   1:L PR[91] 10mm/sec FINE;
   1:  PR[GP1:91,1] = PR[GP1:90,1] + 93.609;
   1:  PR[GP1:91,2] = PR[GP1:90,2] + 108.231;
   1:L PR[91] 10mm/sec FINE;
   1:  PR[GP1:91,1] = PR[GP1:90,1] + 93.731;
   1:  PR[GP1:91,2] = PR[GP1:90,2] + 108.362;
   1:L PR[91] 10mm/sec FINE;
   1:  PR[GP1:91,1] = PR[GP1:90,1] + 93.913;
   1:  PR[GP1:91,2] = PR[GP1:90,2] + 108.511;
   1:L PR[91] 10mm/sec FINE;
   1:  PR[GP1:91,1] = PR[GP1:90,1] + 94.171;
   1:  PR[GP1:91,2] = PR[GP1:90,2] + 108.665;
   1:L PR[91] 10mm/sec FINE;
   1:  PR[GP1:91,1] = PR[GP1:90,1] + 94.322;
   1:  PR[GP1:91,2] = PR[GP1:90,2] + 108.701;
   1:L PR[91] 10mm/sec FINE;
   1:  PR[GP1:91,1] = PR[GP1:90,1] + 94.513;
   1:  PR[GP1:91,2] = PR[GP1:90,2] + 108.801;
   1:L PR[91] 10mm/sec FINE;
   1:  PR[GP1:91,1] = PR[GP1:90,1] + 94.701;
   1:  PR[GP1:91,2] = PR[GP1:90,2] + 108.857;
   1:L PR[91] 10mm/sec FINE;
   1:  PR[GP1:91,1] = PR[GP1:90,1] + 94.821;
   1:  PR[GP1:91,2] = PR[GP1:90,2] + 108.845;
   1:L PR[91] 10mm/sec FINE;
   1:  PR[GP1:91,1] = PR[GP1:90,1] + 95.615;
   1:  PR[GP1:91,2] = PR[GP1:90,2] + 108.874;
   1:L PR[91] 10mm/sec FINE;
   1:  PR[GP1:91,1] = PR[GP1:90,1] + 95.743;
   1:  PR[GP1:91,2] = PR[GP1:90,2] + 108.844;
   1:L PR[91] 10mm/sec FINE;
   1:  PR[GP1:91,1] = PR[GP1:90,1] + 96.602;
   1:  PR[GP1:91,2] = PR[GP1:90,2] + 108.491;
   1:L PR[91] 10mm/sec FINE;
   1:  PR[GP1:91,1] = PR[GP1:90,1] + 96.918;
   1:  PR[GP1:91,2] = PR[GP1:90,2] + 108.237;
   1:L PR[91] 10mm/sec FINE;
   1:  PR[GP1:91,1] = PR[GP1:90,1] + 97.426;
   1:  PR[GP1:91,2] = PR[GP1:90,2] + 107.738;
   1:L PR[91] 10mm/sec FINE;
   1:  PR[GP1:91,1] = PR[GP1:90,1] + 97.882;
   1:  PR[GP1:91,2] = PR[GP1:90,2] + 106.699;
   1:L PR[91] 10mm/sec FINE;
   1:  PR[GP1:91,1] = PR[GP1:90,1] + 98.569;
   1:  PR[GP1:91,2] = PR[GP1:90,2] + 104.056;
   1:L PR[91] 10mm/sec FINE;
   1:  PR[GP1:91,1] = PR[GP1:90,1] + 99.310;
   1:  PR[GP1:91,2] = PR[GP1:90,2] + 102.392;
   1:L PR[91] 10mm/sec FINE;
   1:  PR[GP1:91,1] = PR[GP1:90,1] + 99.684;
   1:  PR[GP1:91,2] = PR[GP1:90,2] + 101.561;
   1:L PR[91] 10mm/sec FINE;
   1:  PR[GP1:91,1] = PR[GP1:90,1] + 101.201;
   1:  PR[GP1:91,2] = PR[GP1:90,2] + 99.269;
   1:L PR[91] 10mm/sec FINE;
   1:  PR[GP1:91,1] = PR[GP1:90,1] + 103.078;
   1:  PR[GP1:91,2] = PR[GP1:90,2] + 97.241;
   1:L PR[91] 10mm/sec FINE;
   1:  PR[GP1:91,1] = PR[GP1:90,1] + 105.216;
   1:  PR[GP1:91,2] = PR[GP1:90,2] + 95.523;
   1:L PR[91] 10mm/sec FINE;
   1:  PR[GP1:91,1] = PR[GP1:90,1] + 107.581;
   1:  PR[GP1:91,2] = PR[GP1:90,2] + 94.152;
   1:L PR[91] 10mm/sec FINE;
   1:  PR[GP1:91,1] = PR[GP1:90,1] + 110.132;
   1:  PR[GP1:91,2] = PR[GP1:90,2] + 93.162;
   1:L PR[91] 10mm/sec FINE;
   1:  PR[GP1:91,1] = PR[GP1:90,1] + 112.809;
   1:  PR[GP1:91,2] = PR[GP1:90,2] + 92.574;
   1:L PR[91] 10mm/sec FINE;
   1:  PR[GP1:91,1] = PR[GP1:90,1] + 115.553;
   1:  PR[GP1:91,2] = PR[GP1:90,2] + 92.397;
   1:L PR[91] 10mm/sec FINE;
   1:  PR[GP1:91,1] = PR[GP1:90,1] + 118.148;
   1:  PR[GP1:91,2] = PR[GP1:90,2] + 92.625;
   1:L PR[91] 10mm/sec FINE;
   1:  PR[GP1:91,1] = PR[GP1:90,1] + 118.473;
   1:  PR[GP1:91,2] = PR[GP1:90,2] + 92.690;
   1:L PR[91] 10mm/sec FINE;
   1:  PR[GP1:91,1] = PR[GP1:90,1] + 120.533;
   1:  PR[GP1:91,2] = PR[GP1:90,2] + 93.200;
   1:L PR[91] 10mm/sec FINE;
   1:  PR[GP1:91,1] = PR[GP1:90,1] + 121.008;
   1:  PR[GP1:91,2] = PR[GP1:90,2] + 93.351;
   1:L PR[91] 10mm/sec FINE;
   1:  PR[GP1:91,1] = PR[GP1:90,1] + 123.294;
   1:  PR[GP1:91,2] = PR[GP1:90,2] + 94.329;
   1:L PR[91] 10mm/sec FINE;
   1:  PR[GP1:91,1] = PR[GP1:90,1] + 123.840;
   1:  PR[GP1:91,2] = PR[GP1:90,2] + 94.647;
   1:L PR[91] 10mm/sec FINE;
   1:  PR[GP1:91,1] = PR[GP1:90,1] + 125.327;
   1:  PR[GP1:91,2] = PR[GP1:90,2] + 95.571;
   1:L PR[91] 10mm/sec FINE;
   1:  PR[GP1:91,1] = PR[GP1:90,1] + 125.920;
   1:  PR[GP1:91,2] = PR[GP1:90,2] + 96.009;
   1:L PR[91] 10mm/sec FINE;
   1:  PR[GP1:91,1] = PR[GP1:90,1] + 127.113;
   1:  PR[GP1:91,2] = PR[GP1:90,2] + 97.040;
   1:L PR[91] 10mm/sec FINE;
   1:  PR[GP1:91,1] = PR[GP1:90,1] + 127.715;
   1:  PR[GP1:91,2] = PR[GP1:90,2] + 97.597;
   1:L PR[91] 10mm/sec FINE;
   1:  PR[GP1:91,1] = PR[GP1:90,1] + 129.232;
   1:  PR[GP1:91,2] = PR[GP1:90,2] + 99.375;
   1:L PR[91] 10mm/sec FINE;
   1:  PR[GP1:91,1] = PR[GP1:90,1] + 129.733;
   1:  PR[GP1:91,2] = PR[GP1:90,2] + 100.102;
   1:L PR[91] 10mm/sec FINE;
   1:  PR[GP1:91,1] = PR[GP1:90,1] + 130.464;
   1:  PR[GP1:91,2] = PR[GP1:90,2] + 101.304;
   1:L PR[91] 10mm/sec FINE;
   1:  PR[GP1:91,1] = PR[GP1:90,1] + 130.906;
   1:  PR[GP1:91,2] = PR[GP1:90,2] + 102.124;
   1:L PR[91] 10mm/sec FINE;
   1:  PR[GP1:91,1] = PR[GP1:90,1] + 131.776;
   1:  PR[GP1:91,2] = PR[GP1:90,2] + 104.258;
   1:L PR[91] 10mm/sec FINE;
   1:  PR[GP1:91,1] = PR[GP1:90,1] + 132.039;
   1:  PR[GP1:91,2] = PR[GP1:90,2] + 105.190;
   1:L PR[91] 10mm/sec FINE;
   1:  PR[GP1:91,1] = PR[GP1:90,1] + 132.341;
   1:  PR[GP1:91,2] = PR[GP1:90,2] + 106.462;
   1:L PR[91] 10mm/sec FINE;
   1:  PR[GP1:91,1] = PR[GP1:90,1] + 132.504;
   1:  PR[GP1:91,2] = PR[GP1:90,2] + 107.439;
   1:L PR[91] 10mm/sec FINE;
   1:  PR[GP1:91,1] = PR[GP1:90,1] + 132.559;
   1:  PR[GP1:91,2] = PR[GP1:90,2] + 108.440;
   1:L PR[91] 10mm/sec FINE;
   1:  PR[GP1:91,1] = PR[GP1:90,1] + 132.683;
   1:  PR[GP1:91,2] = PR[GP1:90,2] + 109.720;
   1:L PR[91] 10mm/sec FINE;
   1:  PR[GP1:91,1] = PR[GP1:90,1] + 132.328;
   1:  PR[GP1:91,2] = PR[GP1:90,2] + 113.118;
   1:L PR[91] 10mm/sec FINE;
   1:  PR[GP1:91,1] = PR[GP1:90,1] + 131.820;
   1:  PR[GP1:91,2] = PR[GP1:90,2] + 114.773;
   1:L PR[91] 10mm/sec FINE;
   1:  PR[GP1:91,1] = PR[GP1:90,1] + 131.524;
   1:  PR[GP1:91,2] = PR[GP1:90,2] + 115.868;
   1:L PR[91] 10mm/sec FINE;
   1:  PR[GP1:91,1] = PR[GP1:90,1] + 131.329;
   1:  PR[GP1:91,2] = PR[GP1:90,2] + 116.382;
   1:L PR[91] 10mm/sec FINE;
   1:  PR[GP1:91,1] = PR[GP1:90,1] + 129.702;
   1:  PR[GP1:91,2] = PR[GP1:90,2] + 119.396;
   1:L PR[91] 10mm/sec FINE;
   1:  PR[GP1:91,1] = PR[GP1:90,1] + 128.498;
   1:  PR[GP1:91,2] = PR[GP1:90,2] + 120.846;
   1:L PR[91] 10mm/sec FINE;
   1:  PR[GP1:91,1] = PR[GP1:90,1] + 128.197;
   1:  PR[GP1:91,2] = PR[GP1:90,2] + 121.262;
   1:L PR[91] 10mm/sec FINE;
   1:  PR[GP1:91,1] = PR[GP1:90,1] + 127.521;
   1:  PR[GP1:91,2] = PR[GP1:90,2] + 122.025;
   1:L PR[91] 10mm/sec FINE;
   1:  PR[GP1:91,1] = PR[GP1:90,1] + 124.860;
   1:  PR[GP1:91,2] = PR[GP1:90,2] + 124.177;
   1:L PR[91] 10mm/sec FINE;
   1:  PR[GP1:91,1] = PR[GP1:90,1] + 121.833;
   1:  PR[GP1:91,2] = PR[GP1:90,2] + 125.763;
   1:L PR[91] 10mm/sec FINE;
   1:  PR[GP1:91,1] = PR[GP1:90,1] + 119.391;
   1:  PR[GP1:91,2] = PR[GP1:90,2] + 126.477;
   1:L PR[91] 10mm/sec FINE;
   1:  PR[GP1:91,1] = PR[GP1:90,1] + 118.835;
   1:  PR[GP1:91,2] = PR[GP1:90,2] + 126.660;
   1:L PR[91] 10mm/sec FINE;
   1:  PR[GP1:91,1] = PR[GP1:90,1] + 118.561;
   1:  PR[GP1:91,2] = PR[GP1:90,2] + 126.721;
   1:L PR[91] 10mm/sec FINE;
   1:  PR[GP1:91,1] = PR[GP1:90,1] + 115.143;
   1:  PR[GP1:91,2] = PR[GP1:90,2] + 127.017;
   1:L PR[91] 10mm/sec FINE;
   1:  PR[GP1:91,1] = PR[GP1:90,1] + 111.751;
   1:  PR[GP1:91,2] = PR[GP1:90,2] + 126.637;
   1:L PR[91] 10mm/sec FINE;
   1:  PR[GP1:91,1] = PR[GP1:90,1] + 108.452;
   1:  PR[GP1:91,2] = PR[GP1:90,2] + 125.593;
   1:L PR[91] 10mm/sec FINE;
   1:  PR[GP1:91,1] = PR[GP1:90,1] + 105.418;
   1:  PR[GP1:91,2] = PR[GP1:90,2] + 123.928;
   1:L PR[91] 10mm/sec FINE;
   1:  PR[GP1:91,1] = PR[GP1:90,1] + 102.775;
   1:  PR[GP1:91,2] = PR[GP1:90,2] + 121.709;
   1:L PR[91] 10mm/sec FINE;
   1:  PR[GP1:91,1] = PR[GP1:90,1] + 100.581;
   1:  PR[GP1:91,2] = PR[GP1:90,2] + 119.016;
   1:L PR[91] 10mm/sec FINE;
   1:  PR[GP1:91,1] = PR[GP1:90,1] + 98.955;
   1:  PR[GP1:91,2] = PR[GP1:90,2] + 115.958;
   1:L PR[91] 10mm/sec FINE;
   1:  PR[GP1:91,1] = PR[GP1:90,1] + 97.961;
   1:  PR[GP1:91,2] = PR[GP1:90,2] + 112.694;
   1:L PR[91] 10mm/sec FINE;
   1:  PR[GP1:91,1] = PR[GP1:90,1] + 97.646;
   1:  PR[GP1:91,2] = PR[GP1:90,2] + 112.056;
   1:L PR[91] 10mm/sec FINE;
   1:  PR[GP1:91,1] = PR[GP1:90,1] + 97.480;
   1:  PR[GP1:91,2] = PR[GP1:90,2] + 111.669;
   1:L PR[91] 10mm/sec FINE;
   1:  PR[GP1:91,1] = PR[GP1:90,1] + 97.077;
   1:  PR[GP1:91,2] = PR[GP1:90,2] + 111.285;
   1:L PR[91] 10mm/sec FINE;
   1:  PR[GP1:91,1] = PR[GP1:90,1] + 96.627;
   1:  PR[GP1:91,2] = PR[GP1:90,2] + 110.927;
   1:L PR[91] 10mm/sec FINE;
   1:  PR[GP1:91,1] = PR[GP1:90,1] + 95.953;
   1:  PR[GP1:91,2] = PR[GP1:90,2] + 110.656;
   1:L PR[91] 10mm/sec FINE;
   1:  PR[GP1:91,1] = PR[GP1:90,1] + 95.474;
   1:  PR[GP1:91,2] = PR[GP1:90,2] + 110.548;
   1:L PR[91] 10mm/sec FINE;
   1:  PR[GP1:91,1] = PR[GP1:90,1] + 94.864;
   1:  PR[GP1:91,2] = PR[GP1:90,2] + 110.569;
   1:L PR[91] 10mm/sec FINE;
   1:  PR[GP1:91,1] = PR[GP1:90,1] + 94.445;
   1:  PR[GP1:91,2] = PR[GP1:90,2] + 110.680;
   1:L PR[91] 10mm/sec FINE;
   1:  PR[GP1:91,1] = PR[GP1:90,1] + 94.027;
   1:  PR[GP1:91,2] = PR[GP1:90,2] + 110.868;
   1:L PR[91] 10mm/sec FINE;
   1:  PR[GP1:91,1] = PR[GP1:90,1] + 93.791;
   1:  PR[GP1:91,2] = PR[GP1:90,2] + 111.065;
   1:L PR[91] 10mm/sec FINE;
   1:  PR[GP1:91,1] = PR[GP1:90,1] + 93.574;
   1:  PR[GP1:91,2] = PR[GP1:90,2] + 111.221;
   1:L PR[91] 10mm/sec FINE;
   1:  PR[GP1:91,1] = PR[GP1:90,1] + 93.370;
   1:  PR[GP1:91,2] = PR[GP1:90,2] + 111.406;
   1:L PR[91] 10mm/sec FINE;
   1:  PR[GP1:91,1] = PR[GP1:90,1] + 93.152;
   1:  PR[GP1:91,2] = PR[GP1:90,2] + 111.677;
   1:L PR[91] 10mm/sec FINE;
   1:  PR[GP1:91,1] = PR[GP1:90,1] + 92.966;
   1:  PR[GP1:91,2] = PR[GP1:90,2] + 112.106;
   1:L PR[91] 10mm/sec FINE;
   1:  PR[GP1:91,1] = PR[GP1:90,1] + 92.851;
   1:  PR[GP1:91,2] = PR[GP1:90,2] + 112.318;
   1:L PR[91] 10mm/sec FINE;
   1:  PR[GP1:91,1] = PR[GP1:90,1] + 92.770;
   1:  PR[GP1:91,2] = PR[GP1:90,2] + 112.528;
   1:L PR[91] 10mm/sec FINE;
   1:  PR[GP1:91,1] = PR[GP1:90,1] + 92.754;
   1:  PR[GP1:91,2] = PR[GP1:90,2] + 112.593;
   1:L PR[91] 10mm/sec FINE;
   1:  PR[GP1:91,1] = PR[GP1:90,1] + 92.675;
   1:  PR[GP1:91,2] = PR[GP1:90,2] + 112.597;
   1:L PR[91] 10mm/sec FINE;
   1:  PR[GP1:91,1] = PR[GP1:90,1] + 92.473;
   1:  PR[GP1:91,2] = PR[GP1:90,2] + 113.514;
   1:L PR[91] 10mm/sec FINE;
   1:  PR[GP1:91,1] = PR[GP1:90,1] + 91.748;
   1:  PR[GP1:91,2] = PR[GP1:90,2] + 116.014;
   1:L PR[91] 10mm/sec FINE;
   1:  PR[GP1:91,1] = PR[GP1:90,1] + 91.367;
   1:  PR[GP1:91,2] = PR[GP1:90,2] + 116.861;
   1:L PR[91] 10mm/sec FINE;
   1:  PR[GP1:91,1] = PR[GP1:90,1] + 90.243;
   1:  PR[GP1:91,2] = PR[GP1:90,2] + 118.946;
   1:L PR[91] 10mm/sec FINE;
   1:  PR[GP1:91,1] = PR[GP1:90,1] + 89.639;
   1:  PR[GP1:91,2] = PR[GP1:90,2] + 119.852;
   1:L PR[91] 10mm/sec FINE;
   1:  PR[GP1:91,1] = PR[GP1:90,1] + 88.262;
   1:  PR[GP1:91,2] = PR[GP1:90,2] + 121.466;
   1:L PR[91] 10mm/sec FINE;
   1:  PR[GP1:91,1] = PR[GP1:90,1] + 87.411;
   1:  PR[GP1:91,2] = PR[GP1:90,2] + 122.375;
   1:L PR[91] 10mm/sec FINE;
   1:  PR[GP1:91,1] = PR[GP1:90,1] + 84.803;
   1:  PR[GP1:91,2] = PR[GP1:90,2] + 124.368;
   1:L PR[91] 10mm/sec FINE;
   1:  PR[GP1:91,1] = PR[GP1:90,1] + 83.575;
   1:  PR[GP1:91,2] = PR[GP1:90,2] + 125.021;
   1:L PR[91] 10mm/sec FINE;
   1:  PR[GP1:91,1] = PR[GP1:90,1] + 81.935;
   1:  PR[GP1:91,2] = PR[GP1:90,2] + 125.795;
   1:L PR[91] 10mm/sec FINE;
   1:  PR[GP1:91,1] = PR[GP1:90,1] + 80.497;
   1:  PR[GP1:91,2] = PR[GP1:90,2] + 126.278;
   1:L PR[91] 10mm/sec FINE;
   1:  PR[GP1:91,1] = PR[GP1:90,1] + 78.911;
   1:  PR[GP1:91,2] = PR[GP1:90,2] + 126.649;
   1:L PR[91] 10mm/sec FINE;
   1:  PR[GP1:91,1] = PR[GP1:90,1] + 77.310;
   1:  PR[GP1:91,2] = PR[GP1:90,2] + 126.906;
   1:L PR[91] 10mm/sec FINE;
   1:  PR[GP1:91,1] = PR[GP1:90,1] + 75.679;
   1:  PR[GP1:91,2] = PR[GP1:90,2] + 126.897;
   1:L PR[91] 10mm/sec FINE;
   1:  PR[GP1:91,1] = PR[GP1:90,1] + 74.111;
   1:  PR[GP1:91,2] = PR[GP1:90,2] + 126.922;
   1:L PR[91] 10mm/sec FINE;
   1:  PR[GP1:91,1] = PR[GP1:90,1] + 72.423;
   1:  PR[GP1:91,2] = PR[GP1:90,2] + 126.632;
   1:L PR[91] 10mm/sec FINE;
   1:  PR[GP1:91,1] = PR[GP1:90,1] + 71.016;
   1:  PR[GP1:91,2] = PR[GP1:90,2] + 126.355;
   1:L PR[91] 10mm/sec FINE;
   1:  PR[GP1:91,1] = PR[GP1:90,1] + 69.332;
   1:  PR[GP1:91,2] = PR[GP1:90,2] + 125.768;
   1:L PR[91] 10mm/sec FINE;
   1:  PR[GP1:91,1] = PR[GP1:90,1] + 68.107;
   1:  PR[GP1:91,2] = PR[GP1:90,2] + 125.242;
   1:L PR[91] 10mm/sec FINE;
   1:  PR[GP1:91,1] = PR[GP1:90,1] + 66.494;
   1:  PR[GP1:91,2] = PR[GP1:90,2] + 124.361;
   1:L PR[91] 10mm/sec FINE;
   1:  PR[GP1:91,1] = PR[GP1:90,1] + 65.466;
   1:  PR[GP1:91,2] = PR[GP1:90,2] + 123.631;
   1:L PR[91] 10mm/sec FINE;
   1:  PR[GP1:91,1] = PR[GP1:90,1] + 63.989;
   1:  PR[GP1:91,2] = PR[GP1:90,2] + 122.474;
   1:L PR[91] 10mm/sec FINE;
   1:  PR[GP1:91,1] = PR[GP1:90,1] + 61.881;
   1:  PR[GP1:91,2] = PR[GP1:90,2] + 120.170;
   1:L PR[91] 10mm/sec FINE;
   1:  PR[GP1:91,1] = PR[GP1:90,1] + 60.844;
   1:  PR[GP1:91,2] = PR[GP1:90,2] + 118.575;
   1:L PR[91] 10mm/sec FINE;
   1:  PR[GP1:91,1] = PR[GP1:90,1] + 60.235;
   1:  PR[GP1:91,2] = PR[GP1:90,2] + 117.535;
   1:L PR[91] 10mm/sec FINE;
   1:  PR[GP1:91,1] = PR[GP1:90,1] + 59.468;
   1:  PR[GP1:91,2] = PR[GP1:90,2] + 115.779;
   1:L PR[91] 10mm/sec FINE;
   1:  PR[GP1:91,1] = PR[GP1:90,1] + 59.094;
   1:  PR[GP1:91,2] = PR[GP1:90,2] + 114.645;
   1:L PR[91] 10mm/sec FINE;
   1:  PR[GP1:91,1] = PR[GP1:90,1] + 58.626;
   1:  PR[GP1:91,2] = PR[GP1:90,2] + 112.789;
   1:L PR[91] 10mm/sec FINE;
   1:  PR[GP1:91,1] = PR[GP1:90,1] + 58.468;
   1:  PR[GP1:91,2] = PR[GP1:90,2] + 110.872;
   1:L PR[91] 10mm/sec FINE;
   1:  PR[GP1:91,1] = PR[GP1:90,1] + 58.343;
   1:  PR[GP1:91,2] = PR[GP1:90,2] + 109.685;
   1:L PR[91] 10mm/sec FINE;
   1:  PR[GP1:91,1] = PR[GP1:90,1] + 58.500;
   1:  PR[GP1:91,2] = PR[GP1:90,2] + 107.787;
   1:L PR[91] 10mm/sec FINE;
   1:  PR[GP1:91,1] = PR[GP1:90,1] + 58.630;
   1:  PR[GP1:91,2] = PR[GP1:90,2] + 106.576;
   1:L PR[91] 10mm/sec FINE;
   1:  PR[GP1:91,1] = PR[GP1:90,1] + 59.091;
   1:  PR[GP1:91,2] = PR[GP1:90,2] + 104.751;
   1:L PR[91] 10mm/sec FINE;
   1:  PR[GP1:91,1] = PR[GP1:90,1] + 59.485;
   1:  PR[GP1:91,2] = PR[GP1:90,2] + 103.554;
   1:L PR[91] 10mm/sec FINE;
   1:  PR[GP1:91,1] = PR[GP1:90,1] + 60.223;
   1:  PR[GP1:91,2] = PR[GP1:90,2] + 101.864;
   1:L PR[91] 10mm/sec FINE;
   1:  PR[GP1:91,1] = PR[GP1:90,1] + 60.899;
   1:  PR[GP1:91,2] = PR[GP1:90,2] + 100.714;
   1:L PR[91] 10mm/sec FINE;
   1:  PR[GP1:91,1] = PR[GP1:90,1] + 61.876;
   1:  PR[GP1:91,2] = PR[GP1:90,2] + 99.212;
   1:L PR[91] 10mm/sec FINE;
   1:  PR[GP1:91,1] = PR[GP1:90,1] + 64.014;
   1:  PR[GP1:91,2] = PR[GP1:90,2] + 96.881;
   1:L PR[91] 10mm/sec FINE;
   1:  PR[GP1:91,1] = PR[GP1:90,1] + 65.370;
   1:  PR[GP1:91,2] = PR[GP1:90,2] + 95.818;
   1:L PR[91] 10mm/sec FINE;
   1:  PR[GP1:91,1] = PR[GP1:90,1] + 66.580;
   1:  PR[GP1:91,2] = PR[GP1:90,2] + 94.963;
   1:L PR[91] 10mm/sec FINE;
   1:  PR[GP1:91,1] = PR[GP1:90,1] + 67.818;
   1:  PR[GP1:91,2] = PR[GP1:90,2] + 94.288;
   1:  PR[GP1:91,3] = PR[GP1:90,3] + 7.900;
   1:L PR[91] 10mm/sec FINE;
   1:  PR[GP1:91,1] = PR[GP1:90,1] + 69.950;
   1:  PR[GP1:91,2] = PR[GP1:90,2] + 93.380;
   1:L PR[91] 10mm/sec FINE;
   1:  PR[GP1:91,1] = PR[GP1:90,1] + 70.874;
   1:  PR[GP1:91,2] = PR[GP1:90,2] + 93.058;
   1:L PR[91] 10mm/sec FINE;
   1:  PR[GP1:91,1] = PR[GP1:90,1] + 71.846;
   1:  PR[GP1:91,2] = PR[GP1:90,2] + 92.891;
   1:L PR[91] 10mm/sec FINE;
   1:  PR[GP1:91,1] = PR[GP1:90,1] + 74.204;
   1:  PR[GP1:91,2] = PR[GP1:90,2] + 92.431;
   1:L PR[91] 10mm/sec FINE;
   1:  PR[GP1:91,1] = PR[GP1:90,1] + 75.008;
   1:  PR[GP1:91,2] = PR[GP1:90,2] + 92.426;
   1:L PR[91] 10mm/sec FINE;
   1:  PR[GP1:91,1] = PR[GP1:90,1] + 77.695;
   1:  PR[GP1:91,2] = PR[GP1:90,2] + 92.483;
   1:L PR[91] 10mm/sec FINE;
   1:  PR[GP1:91,1] = PR[GP1:90,1] + 78.289;
   1:  PR[GP1:91,2] = PR[GP1:90,2] + 92.578;
   1:L PR[91] 10mm/sec FINE;
   1:  PR[GP1:91,1] = PR[GP1:90,1] + 81.225;
   1:  PR[GP1:91,2] = PR[GP1:90,2] + 93.278;
   1:L PR[91] 10mm/sec FINE;
   1:  PR[GP1:91,1] = PR[GP1:90,1] + 81.585;
   1:  PR[GP1:91,2] = PR[GP1:90,2] + 93.398;
   1:L PR[91] 10mm/sec FINE;
   1:  PR[GP1:91,1] = PR[GP1:90,1] + 84.766;
   1:  PR[GP1:91,2] = PR[GP1:90,2] + 94.925;
   1:L PR[91] 10mm/sec FINE;
   1:  PR[GP1:91,1] = PR[GP1:90,1] + 87.670;
   1:  PR[GP1:91,2] = PR[GP1:90,2] + 97.160;
   1:L PR[91] 10mm/sec FINE;
   1:  PR[GP1:91,1] = PR[GP1:90,1] + 89.969;
   1:  PR[GP1:91,2] = PR[GP1:90,2] + 99.834;
   1:L PR[91] 10mm/sec FINE;
   1:  PR[GP1:91,1] = PR[GP1:90,1] + 90.094;
   1:  PR[GP1:91,2] = PR[GP1:90,2] + 100.009;
   1:L PR[91] 10mm/sec FINE;
   1:  PR[GP1:91,1] = PR[GP1:90,1] + 91.694;
   1:  PR[GP1:91,2] = PR[GP1:90,2] + 102.974;
   1:L PR[91] 10mm/sec FINE;
   1:  PR[GP1:91,1] = PR[GP1:90,1] + 91.822;
   1:  PR[GP1:91,2] = PR[GP1:90,2] + 103.264;
   1:L PR[91] 10mm/sec FINE;
   1:  PR[GP1:91,1] = PR[GP1:90,1] + 92.742;
   1:  PR[GP1:91,2] = PR[GP1:90,2] + 106.472;
   1:L PR[91] 10mm/sec FINE;
   1:  PR[GP1:91,1] = PR[GP1:90,1] + 92.815;
   1:  PR[GP1:91,2] = PR[GP1:90,2] + 106.821;
   1:L PR[91] 10mm/sec FINE;
   1:  PR[GP1:91,1] = PR[GP1:90,1] + 92.862;
   1:  PR[GP1:91,2] = PR[GP1:90,2] + 106.963;
   1:L PR[91] 10mm/sec FINE;
   1:  PR[GP1:91,1] = PR[GP1:90,1] + 92.947;
   1:  PR[GP1:91,2] = PR[GP1:90,2] + 107.131;
   1:L PR[91] 10mm/sec FINE;
   1:  PR[GP1:91,1] = PR[GP1:90,1] + 93.041;
   1:  PR[GP1:91,2] = PR[GP1:90,2] + 107.401;
   1:L PR[91] 10mm/sec FINE;
   1:  PR[GP1:91,1] = PR[GP1:90,1] + 93.208;
   1:  PR[GP1:91,2] = PR[GP1:90,2] + 107.720;
   1:L PR[91] 10mm/sec FINE;
   1:  PR[GP1:91,1] = PR[GP1:90,1] + 93.446;
   1:  PR[GP1:91,2] = PR[GP1:90,2] + 108.039;
   1:L PR[91] 10mm/sec FINE;
   1:  PR[GP1:91,1] = PR[GP1:90,1] + 93.610;
   1:  PR[GP1:91,2] = PR[GP1:90,2] + 108.199;
   1:L PR[91] 10mm/sec FINE;
   1:  PR[GP1:91,1] = PR[GP1:90,1] + 93.786;
   1:  PR[GP1:91,2] = PR[GP1:90,2] + 108.282;
   1:L PR[91] 10mm/sec FINE;
   1:  PR[GP1:91,1] = PR[GP1:90,1] + 94.370;
   1:  PR[GP1:91,2] = PR[GP1:90,2] + 108.653;
   1:L PR[91] 10mm/sec FINE;
   1:  PR[GP1:91,1] = PR[GP1:90,1] + 94.818;
   1:  PR[GP1:91,2] = PR[GP1:90,2] + 108.692;
   1:L PR[91] 10mm/sec FINE;
   1:  PR[GP1:91,1] = PR[GP1:90,1] + 95.314;
   1:  PR[GP1:91,2] = PR[GP1:90,2] + 108.764;
   1:L PR[91] 10mm/sec FINE;
   1:  PR[GP1:91,1] = PR[GP1:90,1] + 95.891;
   1:  PR[GP1:91,2] = PR[GP1:90,2] + 108.587;
   1:L PR[91] 10mm/sec FINE;
   1:  PR[GP1:91,1] = PR[GP1:90,1] + 96.258;
   1:  PR[GP1:91,2] = PR[GP1:90,2] + 108.434;
   1:L PR[91] 10mm/sec FINE;
   1:  PR[GP1:91,1] = PR[GP1:90,1] + 96.430;
   1:  PR[GP1:91,2] = PR[GP1:90,2] + 108.316;
   1:L PR[91] 10mm/sec FINE;
   1:  PR[GP1:91,1] = PR[GP1:90,1] + 96.886;
   1:  PR[GP1:91,2] = PR[GP1:90,2] + 107.867;
   1:L PR[91] 10mm/sec FINE;
   1:  PR[GP1:91,1] = PR[GP1:90,1] + 97.040;
   1:  PR[GP1:91,2] = PR[GP1:90,2] + 107.686;
   1:L PR[91] 10mm/sec FINE;
   1:  PR[GP1:91,1] = PR[GP1:90,1] + 97.119;
   1:  PR[GP1:91,2] = PR[GP1:90,2] + 107.556;
   1:L PR[91] 10mm/sec FINE;
   1:  PR[GP1:91,1] = PR[GP1:90,1] + 97.419;
   1:  PR[GP1:91,2] = PR[GP1:90,2] + 106.817;
   1:L PR[91] 10mm/sec FINE;
   1:  PR[GP1:91,1] = PR[GP1:90,1] + 98.137;
   1:  PR[GP1:91,2] = PR[GP1:90,2] + 104.025;
   1:L PR[91] 10mm/sec FINE;
   1:  PR[GP1:91,1] = PR[GP1:90,1] + 99.268;
   1:  PR[GP1:91,2] = PR[GP1:90,2] + 101.523;
   1:L PR[91] 10mm/sec FINE;
   1:  PR[GP1:91,1] = PR[GP1:90,1] + 100.820;
   1:  PR[GP1:91,2] = PR[GP1:90,2] + 99.224;
   1:L PR[91] 10mm/sec FINE;
   1:  PR[GP1:91,1] = PR[GP1:90,1] + 102.722;
   1:  PR[GP1:91,2] = PR[GP1:90,2] + 97.186;
   1:L PR[91] 10mm/sec FINE;
   1:  PR[GP1:91,1] = PR[GP1:90,1] + 104.917;
   1:  PR[GP1:91,2] = PR[GP1:90,2] + 95.464;
   1:L PR[91] 10mm/sec FINE;
   1:  PR[GP1:91,1] = PR[GP1:90,1] + 107.364;
   1:  PR[GP1:91,2] = PR[GP1:90,2] + 94.099;
   1:L PR[91] 10mm/sec FINE;
   1:  PR[GP1:91,1] = PR[GP1:90,1] + 109.942;
   1:  PR[GP1:91,2] = PR[GP1:90,2] + 93.112;
   1:L PR[91] 10mm/sec FINE;
   1:  PR[GP1:91,1] = PR[GP1:90,1] + 112.624;
   1:  PR[GP1:91,2] = PR[GP1:90,2] + 92.526;
   1:L PR[91] 10mm/sec FINE;
   1:  PR[GP1:91,1] = PR[GP1:90,1] + 115.365;
   1:  PR[GP1:91,2] = PR[GP1:90,2] + 92.357;
   1:L PR[91] 10mm/sec FINE;
   1:  PR[GP1:91,1] = PR[GP1:90,1] + 118.099;
   1:  PR[GP1:91,2] = PR[GP1:90,2] + 92.608;
   1:L PR[91] 10mm/sec FINE;
   1:  PR[GP1:91,1] = PR[GP1:90,1] + 120.762;
   1:  PR[GP1:91,2] = PR[GP1:90,2] + 93.274;
   1:L PR[91] 10mm/sec FINE;
   1:  PR[GP1:91,1] = PR[GP1:90,1] + 123.260;
   1:  PR[GP1:91,2] = PR[GP1:90,2] + 94.330;
   1:L PR[91] 10mm/sec FINE;
   1:  PR[GP1:91,1] = PR[GP1:90,1] + 123.348;
   1:  PR[GP1:91,2] = PR[GP1:90,2] + 94.381;
   1:L PR[91] 10mm/sec FINE;
   1:  PR[GP1:91,1] = PR[GP1:90,1] + 125.458;
   1:  PR[GP1:91,2] = PR[GP1:90,2] + 95.691;
   1:L PR[91] 10mm/sec FINE;
   1:  PR[GP1:91,1] = PR[GP1:90,1] + 125.659;
   1:  PR[GP1:91,2] = PR[GP1:90,2] + 95.840;
   1:L PR[91] 10mm/sec FINE;
   1:  PR[GP1:91,1] = PR[GP1:90,1] + 127.353;
   1:  PR[GP1:91,2] = PR[GP1:90,2] + 97.303;
   1:L PR[91] 10mm/sec FINE;
   1:  PR[GP1:91,1] = PR[GP1:90,1] + 127.623;
   1:  PR[GP1:91,2] = PR[GP1:90,2] + 97.552;
   1:L PR[91] 10mm/sec FINE;
   1:  PR[GP1:91,1] = PR[GP1:90,1] + 129.253;
   1:  PR[GP1:91,2] = PR[GP1:90,2] + 99.473;
   1:L PR[91] 10mm/sec FINE;
   1:  PR[GP1:91,1] = PR[GP1:90,1] + 129.513;
   1:  PR[GP1:91,2] = PR[GP1:90,2] + 99.850;
   1:L PR[91] 10mm/sec FINE;
   1:  PR[GP1:91,1] = PR[GP1:90,1] + 130.550;
   1:  PR[GP1:91,2] = PR[GP1:90,2] + 101.556;
   1:L PR[91] 10mm/sec FINE;
   1:  PR[GP1:91,1] = PR[GP1:90,1] + 130.800;
   1:  PR[GP1:91,2] = PR[GP1:90,2] + 102.020;
   1:L PR[91] 10mm/sec FINE;
   1:  PR[GP1:91,1] = PR[GP1:90,1] + 131.736;
   1:  PR[GP1:91,2] = PR[GP1:90,2] + 104.309;
   1:L PR[91] 10mm/sec FINE;
   1:  PR[GP1:91,1] = PR[GP1:90,1] + 131.893;
   1:  PR[GP1:91,2] = PR[GP1:90,2] + 104.866;
   1:L PR[91] 10mm/sec FINE;
   1:  PR[GP1:91,1] = PR[GP1:90,1] + 132.322;
   1:  PR[GP1:91,2] = PR[GP1:90,2] + 106.672;
   1:L PR[91] 10mm/sec FINE;
   1:  PR[GP1:91,1] = PR[GP1:90,1] + 132.423;
   1:  PR[GP1:91,2] = PR[GP1:90,2] + 107.274;
   1:L PR[91] 10mm/sec FINE;
   1:  PR[GP1:91,1] = PR[GP1:90,1] + 132.457;
   1:  PR[GP1:91,2] = PR[GP1:90,2] + 107.895;
   1:L PR[91] 10mm/sec FINE;
   1:  PR[GP1:91,1] = PR[GP1:90,1] + 132.633;
   1:  PR[GP1:91,2] = PR[GP1:90,2] + 109.715;
   1:L PR[91] 10mm/sec FINE;
   1:  PR[GP1:91,1] = PR[GP1:90,1] + 132.271;
   1:  PR[GP1:91,2] = PR[GP1:90,2] + 113.112;
   1:L PR[91] 10mm/sec FINE;
   1:  PR[GP1:91,1] = PR[GP1:90,1] + 131.549;
   1:  PR[GP1:91,2] = PR[GP1:90,2] + 115.464;
   1:L PR[91] 10mm/sec FINE;
   1:  PR[GP1:91,1] = PR[GP1:90,1] + 131.380;
   1:  PR[GP1:91,2] = PR[GP1:90,2] + 116.091;
   1:L PR[91] 10mm/sec FINE;
   1:  PR[GP1:91,1] = PR[GP1:90,1] + 131.271;
   1:  PR[GP1:91,2] = PR[GP1:90,2] + 116.377;
   1:L PR[91] 10mm/sec FINE;
   1:  PR[GP1:91,1] = PR[GP1:90,1] + 129.643;
   1:  PR[GP1:91,2] = PR[GP1:90,2] + 119.392;
   1:L PR[91] 10mm/sec FINE;
   1:  PR[GP1:91,1] = PR[GP1:90,1] + 127.934;
   1:  PR[GP1:91,2] = PR[GP1:90,2] + 121.449;
   1:L PR[91] 10mm/sec FINE;
   1:  PR[GP1:91,1] = PR[GP1:90,1] + 127.786;
   1:  PR[GP1:91,2] = PR[GP1:90,2] + 121.654;
   1:L PR[91] 10mm/sec FINE;
   1:  PR[GP1:91,1] = PR[GP1:90,1] + 127.461;
   1:  PR[GP1:91,2] = PR[GP1:90,2] + 122.020;
   1:L PR[91] 10mm/sec FINE;
   1:  PR[GP1:91,1] = PR[GP1:90,1] + 124.800;
   1:  PR[GP1:91,2] = PR[GP1:90,2] + 124.172;
   1:L PR[91] 10mm/sec FINE;
   1:  PR[GP1:91,1] = PR[GP1:90,1] + 121.773;
   1:  PR[GP1:91,2] = PR[GP1:90,2] + 125.758;
   1:L PR[91] 10mm/sec FINE;
   1:  PR[GP1:91,1] = PR[GP1:90,1] + 119.646;
   1:  PR[GP1:91,2] = PR[GP1:90,2] + 126.380;
   1:L PR[91] 10mm/sec FINE;
   1:  PR[GP1:91,1] = PR[GP1:90,1] + 118.478;
   1:  PR[GP1:91,2] = PR[GP1:90,2] + 126.715;
   1:L PR[91] 10mm/sec FINE;
   1:  PR[GP1:91,1] = PR[GP1:90,1] + 115.028;
   1:  PR[GP1:91,2] = PR[GP1:90,2] + 127.006;
   1:L PR[91] 10mm/sec FINE;
   1:  PR[GP1:91,1] = PR[GP1:90,1] + 111.577;
   1:  PR[GP1:91,2] = PR[GP1:90,2] + 126.621;
   1:L PR[91] 10mm/sec FINE;
   1:  PR[GP1:91,1] = PR[GP1:90,1] + 108.270;
   1:  PR[GP1:91,2] = PR[GP1:90,2] + 125.575;
   1:L PR[91] 10mm/sec FINE;
   1:  PR[GP1:91,1] = PR[GP1:90,1] + 105.227;
   1:  PR[GP1:91,2] = PR[GP1:90,2] + 123.908;
   1:L PR[91] 10mm/sec FINE;
   1:  PR[GP1:91,1] = PR[GP1:90,1] + 102.512;
   1:  PR[GP1:91,2] = PR[GP1:90,2] + 121.681;
   1:L PR[91] 10mm/sec FINE;
   1:  PR[GP1:91,1] = PR[GP1:90,1] + 100.969;
   1:  PR[GP1:91,2] = PR[GP1:90,2] + 119.802;
   1:L PR[91] 10mm/sec FINE;
   1:  PR[GP1:91,1] = PR[GP1:90,1] + 100.277;
   1:  PR[GP1:91,2] = PR[GP1:90,2] + 118.983;
   1:L PR[91] 10mm/sec FINE;
   1:  PR[GP1:91,1] = PR[GP1:90,1] + 98.595;
   1:  PR[GP1:91,2] = PR[GP1:90,2] + 115.919;
   1:L PR[91] 10mm/sec FINE;
   1:  PR[GP1:91,1] = PR[GP1:90,1] + 97.578;
   1:  PR[GP1:91,2] = PR[GP1:90,2] + 112.683;
   1:L PR[91] 10mm/sec FINE;
   1:  PR[GP1:91,1] = PR[GP1:90,1] + 97.157;
   1:  PR[GP1:91,2] = PR[GP1:90,2] + 111.737;
   1:L PR[91] 10mm/sec FINE;
   1:  PR[GP1:91,1] = PR[GP1:90,1] + 96.424;
   1:  PR[GP1:91,2] = PR[GP1:90,2] + 111.035;
   1:L PR[91] 10mm/sec FINE;
   1:  PR[GP1:91,1] = PR[GP1:90,1] + 96.066;
   1:  PR[GP1:91,2] = PR[GP1:90,2] + 110.840;
   1:L PR[91] 10mm/sec FINE;
   1:  PR[GP1:91,1] = PR[GP1:90,1] + 95.723;
   1:  PR[GP1:91,2] = PR[GP1:90,2] + 110.736;
   1:L PR[91] 10mm/sec FINE;
   1:  PR[GP1:91,1] = PR[GP1:90,1] + 95.100;
   1:  PR[GP1:91,2] = PR[GP1:90,2] + 110.625;
   1:L PR[91] 10mm/sec FINE;
   1:  PR[GP1:91,1] = PR[GP1:90,1] + 94.689;
   1:  PR[GP1:91,2] = PR[GP1:90,2] + 110.745;
   1:L PR[91] 10mm/sec FINE;
   1:  PR[GP1:91,1] = PR[GP1:90,1] + 94.191;
   1:  PR[GP1:91,2] = PR[GP1:90,2] + 110.833;
   1:L PR[91] 10mm/sec FINE;
   1:  PR[GP1:91,1] = PR[GP1:90,1] + 93.792;
   1:  PR[GP1:91,2] = PR[GP1:90,2] + 111.065;
   1:L PR[91] 10mm/sec FINE;
   1:  PR[GP1:91,1] = PR[GP1:90,1] + 93.446;
   1:  PR[GP1:91,2] = PR[GP1:90,2] + 111.389;
   1:L PR[91] 10mm/sec FINE;
   1:  PR[GP1:91,1] = PR[GP1:90,1] + 93.211;
   1:  PR[GP1:91,2] = PR[GP1:90,2] + 111.692;
   1:L PR[91] 10mm/sec FINE;
   1:  PR[GP1:91,1] = PR[GP1:90,1] + 92.975;
   1:  PR[GP1:91,2] = PR[GP1:90,2] + 112.157;
   1:L PR[91] 10mm/sec FINE;
   1:  PR[GP1:91,1] = PR[GP1:90,1] + 92.865;
   1:  PR[GP1:91,2] = PR[GP1:90,2] + 112.441;
   1:L PR[91] 10mm/sec FINE;
   1:  PR[GP1:91,1] = PR[GP1:90,1] + 92.828;
   1:  PR[GP1:91,2] = PR[GP1:90,2] + 112.589;
   1:L PR[91] 10mm/sec FINE;
   1:  PR[GP1:91,1] = PR[GP1:90,1] + 92.783;
   1:  PR[GP1:91,2] = PR[GP1:90,2] + 112.592;
   1:L PR[91] 10mm/sec FINE;
   1:  PR[GP1:91,1] = PR[GP1:90,1] + 91.725;
   1:  PR[GP1:91,2] = PR[GP1:90,2] + 116.217;
   1:L PR[91] 10mm/sec FINE;
   1:  PR[GP1:91,1] = PR[GP1:90,1] + 90.075;
   1:  PR[GP1:91,2] = PR[GP1:90,2] + 119.298;
   1:L PR[91] 10mm/sec FINE;
   1:  PR[GP1:91,1] = PR[GP1:90,1] + 89.881;
   1:  PR[GP1:91,2] = PR[GP1:90,2] + 119.590;
   1:L PR[91] 10mm/sec FINE;
   1:  PR[GP1:91,1] = PR[GP1:90,1] + 87.926;
   1:  PR[GP1:91,2] = PR[GP1:90,2] + 121.881;
   1:L PR[91] 10mm/sec FINE;
   1:  PR[GP1:91,1] = PR[GP1:90,1] + 87.535;
   1:  PR[GP1:91,2] = PR[GP1:90,2] + 122.299;
   1:L PR[91] 10mm/sec FINE;
   1:  PR[GP1:91,1] = PR[GP1:90,1] + 84.781;
   1:  PR[GP1:91,2] = PR[GP1:90,2] + 124.402;
   1:L PR[91] 10mm/sec FINE;
   1:  PR[GP1:91,1] = PR[GP1:90,1] + 84.094;
   1:  PR[GP1:91,2] = PR[GP1:90,2] + 124.767;
   1:L PR[91] 10mm/sec FINE;
   1:  PR[GP1:91,1] = PR[GP1:90,1] + 81.765;
   1:  PR[GP1:91,2] = PR[GP1:90,2] + 125.868;
   1:L PR[91] 10mm/sec FINE;
   1:  PR[GP1:91,1] = PR[GP1:90,1] + 80.856;
   1:  PR[GP1:91,2] = PR[GP1:90,2] + 126.172;
   1:L PR[91] 10mm/sec FINE;
   1:  PR[GP1:91,1] = PR[GP1:90,1] + 78.603;
   1:  PR[GP1:91,2] = PR[GP1:90,2] + 126.700;
   1:L PR[91] 10mm/sec FINE;
   1:  PR[GP1:91,1] = PR[GP1:90,1] + 77.509;
   1:  PR[GP1:91,2] = PR[GP1:90,2] + 126.875;
   1:L PR[91] 10mm/sec FINE;
   1:  PR[GP1:91,1] = PR[GP1:90,1] + 76.392;
   1:  PR[GP1:91,2] = PR[GP1:90,2] + 126.869;
   1:L PR[91] 10mm/sec FINE;
   1:  PR[GP1:91,1] = PR[GP1:90,1] + 74.165;
   1:  PR[GP1:91,2] = PR[GP1:90,2] + 126.905;
   1:L PR[91] 10mm/sec FINE;
   1:  PR[GP1:91,1] = PR[GP1:90,1] + 72.948;
   1:  PR[GP1:91,2] = PR[GP1:90,2] + 126.695;
   1:L PR[91] 10mm/sec FINE;
   1:  PR[GP1:91,1] = PR[GP1:90,1] + 70.947;
   1:  PR[GP1:91,2] = PR[GP1:90,2] + 126.301;
   1:L PR[91] 10mm/sec FINE;
   1:  PR[GP1:91,1] = PR[GP1:90,1] + 69.687;
   1:  PR[GP1:91,2] = PR[GP1:90,2] + 125.862;
   1:L PR[91] 10mm/sec FINE;
   1:  PR[GP1:91,1] = PR[GP1:90,1] + 67.945;
   1:  PR[GP1:91,2] = PR[GP1:90,2] + 125.114;
   1:L PR[91] 10mm/sec FINE;
   1:  PR[GP1:91,1] = PR[GP1:90,1] + 66.706;
   1:  PR[GP1:91,2] = PR[GP1:90,2] + 124.438;
   1:L PR[91] 10mm/sec FINE;
   1:  PR[GP1:91,1] = PR[GP1:90,1] + 65.244;
   1:  PR[GP1:91,2] = PR[GP1:90,2] + 123.399;
   1:L PR[91] 10mm/sec FINE;
   1:  PR[GP1:91,1] = PR[GP1:90,1] + 64.089;
   1:  PR[GP1:91,2] = PR[GP1:90,2] + 122.494;
   1:L PR[91] 10mm/sec FINE;
   1:  PR[GP1:91,1] = PR[GP1:90,1] + 61.904;
   1:  PR[GP1:91,2] = PR[GP1:90,2] + 120.106;
   1:L PR[91] 10mm/sec FINE;
   1:  PR[GP1:91,1] = PR[GP1:90,1] + 61.084;
   1:  PR[GP1:91,2] = PR[GP1:90,2] + 118.845;
   1:L PR[91] 10mm/sec FINE;
   1:  PR[GP1:91,1] = PR[GP1:90,1] + 60.218;
   1:  PR[GP1:91,2] = PR[GP1:90,2] + 117.364;
   1:L PR[91] 10mm/sec FINE;
   1:  PR[GP1:91,1] = PR[GP1:90,1] + 59.608;
   1:  PR[GP1:91,2] = PR[GP1:90,2] + 115.969;
   1:L PR[91] 10mm/sec FINE;
   1:  PR[GP1:91,1] = PR[GP1:90,1] + 59.077;
   1:  PR[GP1:91,2] = PR[GP1:90,2] + 114.356;
   1:L PR[91] 10mm/sec FINE;
   1:  PR[GP1:91,1] = PR[GP1:90,1] + 58.704;
   1:  PR[GP1:91,2] = PR[GP1:90,2] + 112.881;
   1:L PR[91] 10mm/sec FINE;
   1:  PR[GP1:91,1] = PR[GP1:90,1] + 58.578;
   1:  PR[GP1:91,2] = PR[GP1:90,2] + 111.354;
   1:L PR[91] 10mm/sec FINE;
   1:  PR[GP1:91,1] = PR[GP1:90,1] + 58.401;
   1:  PR[GP1:91,2] = PR[GP1:90,2] + 109.666;
   1:L PR[91] 10mm/sec FINE;
   1:  PR[GP1:91,1] = PR[GP1:90,1] + 58.525;
   1:  PR[GP1:91,2] = PR[GP1:90,2] + 108.165;
   1:L PR[91] 10mm/sec FINE;
   1:  PR[GP1:91,1] = PR[GP1:90,1] + 58.711;
   1:  PR[GP1:91,2] = PR[GP1:90,2] + 106.442;
   1:L PR[91] 10mm/sec FINE;
   1:  PR[GP1:91,1] = PR[GP1:90,1] + 59.071;
   1:  PR[GP1:91,2] = PR[GP1:90,2] + 105.012;
   1:L PR[91] 10mm/sec FINE;
   1:  PR[GP1:91,1] = PR[GP1:90,1] + 59.633;
   1:  PR[GP1:91,2] = PR[GP1:90,2] + 103.309;
   1:L PR[91] 10mm/sec FINE;
   1:  PR[GP1:91,1] = PR[GP1:90,1] + 60.201;
   1:  PR[GP1:91,2] = PR[GP1:90,2] + 102.007;
   1:L PR[91] 10mm/sec FINE;
   1:  PR[GP1:91,1] = PR[GP1:90,1] + 61.162;
   1:  PR[GP1:91,2] = PR[GP1:90,2] + 100.372;
   1:L PR[91] 10mm/sec FINE;
   1:  PR[GP1:91,1] = PR[GP1:90,1] + 61.897;
   1:  PR[GP1:91,2] = PR[GP1:90,2] + 99.243;
   1:L PR[91] 10mm/sec FINE;
   1:  PR[GP1:91,1] = PR[GP1:90,1] + 64.124;
   1:  PR[GP1:91,2] = PR[GP1:90,2] + 96.815;
   1:L PR[91] 10mm/sec FINE;
   1:  PR[GP1:91,1] = PR[GP1:90,1] + 65.108;
   1:  PR[GP1:91,2] = PR[GP1:90,2] + 96.044;
   1:L PR[91] 10mm/sec FINE;
   1:  PR[GP1:91,1] = PR[GP1:90,1] + 66.828;
   1:  PR[GP1:91,2] = PR[GP1:90,2] + 94.829;
   1:L PR[91] 10mm/sec FINE;
   1:  PR[GP1:91,1] = PR[GP1:90,1] + 67.619;
   1:  PR[GP1:91,2] = PR[GP1:90,2] + 94.397;
   1:  PR[GP1:91,3] = PR[GP1:90,3] + 8.900;
   1:L PR[91] 10mm/sec FINE;
   1:  PR[GP1:91,1] = PR[GP1:90,1] + 70.382;
   1:  PR[GP1:91,2] = PR[GP1:90,2] + 93.221;
   1:L PR[91] 10mm/sec FINE;
   1:  PR[GP1:91,1] = PR[GP1:90,1] + 70.786;
   1:  PR[GP1:91,2] = PR[GP1:90,2] + 93.080;
   1:L PR[91] 10mm/sec FINE;
   1:  PR[GP1:91,1] = PR[GP1:90,1] + 74.268;
   1:  PR[GP1:91,2] = PR[GP1:90,2] + 92.411;
   1:L PR[91] 10mm/sec FINE;
   1:  PR[GP1:91,1] = PR[GP1:90,1] + 74.468;
   1:  PR[GP1:91,2] = PR[GP1:90,2] + 92.409;
   1:L PR[91] 10mm/sec FINE;
   1:  PR[GP1:91,1] = PR[GP1:90,1] + 77.920;
   1:  PR[GP1:91,2] = PR[GP1:90,2] + 92.478;
   1:L PR[91] 10mm/sec FINE;
   1:  PR[GP1:91,1] = PR[GP1:90,1] + 81.398;
   1:  PR[GP1:91,2] = PR[GP1:90,2] + 93.258;
   1:L PR[91] 10mm/sec FINE;
   1:  PR[GP1:91,1] = PR[GP1:90,1] + 81.771;
   1:  PR[GP1:91,2] = PR[GP1:90,2] + 93.391;
   1:L PR[91] 10mm/sec FINE;
   1:  PR[GP1:91,1] = PR[GP1:90,1] + 84.596;
   1:  PR[GP1:91,2] = PR[GP1:90,2] + 94.698;
   1:L PR[91] 10mm/sec FINE;
   1:  PR[GP1:91,1] = PR[GP1:90,1] + 85.239;
   1:  PR[GP1:91,2] = PR[GP1:90,2] + 95.087;
   1:L PR[91] 10mm/sec FINE;
   1:  PR[GP1:91,1] = PR[GP1:90,1] + 87.414;
   1:  PR[GP1:91,2] = PR[GP1:90,2] + 96.726;
   1:L PR[91] 10mm/sec FINE;
   1:  PR[GP1:91,1] = PR[GP1:90,1] + 88.197;
   1:  PR[GP1:91,2] = PR[GP1:90,2] + 97.451;
   1:L PR[91] 10mm/sec FINE;
   1:  PR[GP1:91,1] = PR[GP1:90,1] + 89.760;
   1:  PR[GP1:91,2] = PR[GP1:90,2] + 99.270;
   1:L PR[91] 10mm/sec FINE;
   1:  PR[GP1:91,1] = PR[GP1:90,1] + 90.521;
   1:  PR[GP1:91,2] = PR[GP1:90,2] + 100.335;
   1:L PR[91] 10mm/sec FINE;
   1:  PR[GP1:91,1] = PR[GP1:90,1] + 91.558;
   1:  PR[GP1:91,2] = PR[GP1:90,2] + 102.257;
   1:L PR[91] 10mm/sec FINE;
   1:  PR[GP1:91,1] = PR[GP1:90,1] + 92.145;
   1:  PR[GP1:91,2] = PR[GP1:90,2] + 103.576;
   1:L PR[91] 10mm/sec FINE;
   1:  PR[GP1:91,1] = PR[GP1:90,1] + 92.720;
   1:  PR[GP1:91,2] = PR[GP1:90,2] + 105.582;
   1:L PR[91] 10mm/sec FINE;
   1:  PR[GP1:91,1] = PR[GP1:90,1] + 92.826;
   1:  PR[GP1:91,2] = PR[GP1:90,2] + 106.123;
   1:L PR[91] 10mm/sec FINE;
   1:  PR[GP1:91,1] = PR[GP1:90,1] + 93.140;
   1:  PR[GP1:91,2] = PR[GP1:90,2] + 106.943;
   1:L PR[91] 10mm/sec FINE;
   1:  PR[GP1:91,1] = PR[GP1:90,1] + 93.284;
   1:  PR[GP1:91,2] = PR[GP1:90,2] + 107.365;
   1:L PR[91] 10mm/sec FINE;
   1:  PR[GP1:91,1] = PR[GP1:90,1] + 93.481;
   1:  PR[GP1:91,2] = PR[GP1:90,2] + 107.527;
   1:L PR[91] 10mm/sec FINE;
   1:  PR[GP1:91,1] = PR[GP1:90,1] + 93.647;
   1:  PR[GP1:91,2] = PR[GP1:90,2] + 107.756;
   1:L PR[91] 10mm/sec FINE;
   1:  PR[GP1:91,1] = PR[GP1:90,1] + 93.995;
   1:  PR[GP1:91,2] = PR[GP1:90,2] + 108.106;
   1:L PR[91] 10mm/sec FINE;
   1:  PR[GP1:91,1] = PR[GP1:90,1] + 94.410;
   1:  PR[GP1:91,2] = PR[GP1:90,2] + 108.197;
   1:L PR[91] 10mm/sec FINE;
   1:  PR[GP1:91,1] = PR[GP1:90,1] + 94.918;
   1:  PR[GP1:91,2] = PR[GP1:90,2] + 108.392;
   1:L PR[91] 10mm/sec FINE;
   1:  PR[GP1:91,1] = PR[GP1:90,1] + 95.727;
   1:  PR[GP1:91,2] = PR[GP1:90,2] + 108.243;
   1:L PR[91] 10mm/sec FINE;
   1:  PR[GP1:91,1] = PR[GP1:90,1] + 95.990;
   1:  PR[GP1:91,2] = PR[GP1:90,2] + 108.143;
   1:L PR[91] 10mm/sec FINE;
   1:  PR[GP1:91,1] = PR[GP1:90,1] + 96.596;
   1:  PR[GP1:91,2] = PR[GP1:90,2] + 107.540;
   1:L PR[91] 10mm/sec FINE;
   1:  PR[GP1:91,1] = PR[GP1:90,1] + 96.841;
   1:  PR[GP1:91,2] = PR[GP1:90,2] + 107.126;
   1:L PR[91] 10mm/sec FINE;
   1:  PR[GP1:91,1] = PR[GP1:90,1] + 96.945;
   1:  PR[GP1:91,2] = PR[GP1:90,2] + 106.892;
   1:L PR[91] 10mm/sec FINE;
   1:  PR[GP1:91,1] = PR[GP1:90,1] + 97.684;
   1:  PR[GP1:91,2] = PR[GP1:90,2] + 103.988;
   1:L PR[91] 10mm/sec FINE;
   1:  PR[GP1:91,1] = PR[GP1:90,1] + 98.812;
   1:  PR[GP1:91,2] = PR[GP1:90,2] + 101.474;
   1:L PR[91] 10mm/sec FINE;
   1:  PR[GP1:91,1] = PR[GP1:90,1] + 100.364;
   1:  PR[GP1:91,2] = PR[GP1:90,2] + 99.163;
   1:L PR[91] 10mm/sec FINE;
   1:  PR[GP1:91,1] = PR[GP1:90,1] + 102.299;
   1:  PR[GP1:91,2] = PR[GP1:90,2] + 97.120;
   1:L PR[91] 10mm/sec FINE;
   1:  PR[GP1:91,1] = PR[GP1:90,1] + 104.563;
   1:  PR[GP1:91,2] = PR[GP1:90,2] + 95.397;
   1:L PR[91] 10mm/sec FINE;
   1:  PR[GP1:91,1] = PR[GP1:90,1] + 107.030;
   1:  PR[GP1:91,2] = PR[GP1:90,2] + 94.028;
   1:L PR[91] 10mm/sec FINE;
   1:  PR[GP1:91,1] = PR[GP1:90,1] + 109.677;
   1:  PR[GP1:91,2] = PR[GP1:90,2] + 93.049;
   1:L PR[91] 10mm/sec FINE;
   1:  PR[GP1:91,1] = PR[GP1:90,1] + 112.438;
   1:  PR[GP1:91,2] = PR[GP1:90,2] + 92.478;
   1:L PR[91] 10mm/sec FINE;
   1:  PR[GP1:91,1] = PR[GP1:90,1] + 115.183;
   1:  PR[GP1:91,2] = PR[GP1:90,2] + 92.312;
   1:L PR[91] 10mm/sec FINE;
   1:  PR[GP1:91,1] = PR[GP1:90,1] + 117.921;
   1:  PR[GP1:91,2] = PR[GP1:90,2] + 92.566;
   1:L PR[91] 10mm/sec FINE;
   1:  PR[GP1:91,1] = PR[GP1:90,1] + 120.586;
   1:  PR[GP1:91,2] = PR[GP1:90,2] + 93.235;
   1:L PR[91] 10mm/sec FINE;
   1:  PR[GP1:91,1] = PR[GP1:90,1] + 123.114;
   1:  PR[GP1:91,2] = PR[GP1:90,2] + 94.301;
   1:L PR[91] 10mm/sec FINE;
   1:  PR[GP1:91,1] = PR[GP1:90,1] + 125.444;
   1:  PR[GP1:91,2] = PR[GP1:90,2] + 95.739;
   1:L PR[91] 10mm/sec FINE;
   1:  PR[GP1:91,1] = PR[GP1:90,1] + 127.521;
   1:  PR[GP1:91,2] = PR[GP1:90,2] + 97.514;
   1:L PR[91] 10mm/sec FINE;
   1:  PR[GP1:91,1] = PR[GP1:90,1] + 129.271;
   1:  PR[GP1:91,2] = PR[GP1:90,2] + 99.568;
   1:L PR[91] 10mm/sec FINE;
   1:  PR[GP1:91,1] = PR[GP1:90,1] + 130.696;
   1:  PR[GP1:91,2] = PR[GP1:90,2] + 101.921;
   1:L PR[91] 10mm/sec FINE;
   1:  PR[GP1:91,1] = PR[GP1:90,1] + 131.695;
   1:  PR[GP1:91,2] = PR[GP1:90,2] + 104.357;
   1:L PR[91] 10mm/sec FINE;
   1:  PR[GP1:91,1] = PR[GP1:90,1] + 132.304;
   1:  PR[GP1:91,2] = PR[GP1:90,2] + 106.882;
   1:L PR[91] 10mm/sec FINE;
   1:  PR[GP1:91,1] = PR[GP1:90,1] + 132.342;
   1:  PR[GP1:91,2] = PR[GP1:90,2] + 107.112;
   1:L PR[91] 10mm/sec FINE;
   1:  PR[GP1:91,1] = PR[GP1:90,1] + 132.572;
   1:  PR[GP1:91,2] = PR[GP1:90,2] + 109.708;
   1:L PR[91] 10mm/sec FINE;
   1:  PR[GP1:91,1] = PR[GP1:90,1] + 132.214;
   1:  PR[GP1:91,2] = PR[GP1:90,2] + 113.108;
   1:L PR[91] 10mm/sec FINE;
   1:  PR[GP1:91,1] = PR[GP1:90,1] + 131.210;
   1:  PR[GP1:91,2] = PR[GP1:90,2] + 116.378;
   1:L PR[91] 10mm/sec FINE;
   1:  PR[GP1:91,1] = PR[GP1:90,1] + 129.584;
   1:  PR[GP1:91,2] = PR[GP1:90,2] + 119.387;
   1:L PR[91] 10mm/sec FINE;
   1:  PR[GP1:91,1] = PR[GP1:90,1] + 127.397;
   1:  PR[GP1:91,2] = PR[GP1:90,2] + 122.017;
   1:L PR[91] 10mm/sec FINE;
   1:  PR[GP1:91,1] = PR[GP1:90,1] + 124.702;
   1:  PR[GP1:91,2] = PR[GP1:90,2] + 124.164;
   1:L PR[91] 10mm/sec FINE;
   1:  PR[GP1:91,1] = PR[GP1:90,1] + 121.630;
   1:  PR[GP1:91,2] = PR[GP1:90,2] + 125.745;
   1:L PR[91] 10mm/sec FINE;
   1:  PR[GP1:91,1] = PR[GP1:90,1] + 118.301;
   1:  PR[GP1:91,2] = PR[GP1:90,2] + 126.700;
   1:L PR[91] 10mm/sec FINE;
   1:  PR[GP1:91,1] = PR[GP1:90,1] + 114.842;
   1:  PR[GP1:91,2] = PR[GP1:90,2] + 126.989;
   1:L PR[91] 10mm/sec FINE;
   1:  PR[GP1:91,1] = PR[GP1:90,1] + 111.398;
   1:  PR[GP1:91,2] = PR[GP1:90,2] + 126.604;
   1:L PR[91] 10mm/sec FINE;
   1:  PR[GP1:91,1] = PR[GP1:90,1] + 108.060;
   1:  PR[GP1:91,2] = PR[GP1:90,2] + 125.554;
   1:L PR[91] 10mm/sec FINE;
   1:  PR[GP1:91,1] = PR[GP1:90,1] + 104.943;
   1:  PR[GP1:91,2] = PR[GP1:90,2] + 123.879;
   1:L PR[91] 10mm/sec FINE;
   1:  PR[GP1:91,1] = PR[GP1:90,1] + 103.404;
   1:  PR[GP1:91,2] = PR[GP1:90,2] + 122.616;
   1:L PR[91] 10mm/sec FINE;
   1:  PR[GP1:91,1] = PR[GP1:90,1] + 102.191;
   1:  PR[GP1:91,2] = PR[GP1:90,2] + 121.647;
   1:L PR[91] 10mm/sec FINE;
   1:  PR[GP1:91,1] = PR[GP1:90,1] + 99.910;
   1:  PR[GP1:91,2] = PR[GP1:90,2] + 118.944;
   1:L PR[91] 10mm/sec FINE;
   1:  PR[GP1:91,1] = PR[GP1:90,1] + 98.183;
   1:  PR[GP1:91,2] = PR[GP1:90,2] + 115.869;
   1:L PR[91] 10mm/sec FINE;
   1:  PR[GP1:91,1] = PR[GP1:90,1] + 97.146;
   1:  PR[GP1:91,2] = PR[GP1:90,2] + 112.670;
   1:L PR[91] 10mm/sec FINE;
   1:  PR[GP1:91,1] = PR[GP1:90,1] + 97.047;
   1:  PR[GP1:91,2] = PR[GP1:90,2] + 112.447;
   1:L PR[91] 10mm/sec FINE;
   1:  PR[GP1:91,1] = PR[GP1:90,1] + 96.995;
   1:  PR[GP1:91,2] = PR[GP1:90,2] + 112.247;
   1:L PR[91] 10mm/sec FINE;
   1:  PR[GP1:91,1] = PR[GP1:90,1] + 96.887;
   1:  PR[GP1:91,2] = PR[GP1:90,2] + 111.994;
   1:L PR[91] 10mm/sec FINE;
   1:  PR[GP1:91,1] = PR[GP1:90,1] + 96.663;
   1:  PR[GP1:91,2] = PR[GP1:90,2] + 111.662;
   1:L PR[91] 10mm/sec FINE;
   1:  PR[GP1:91,1] = PR[GP1:90,1] + 95.969;
   1:  PR[GP1:91,2] = PR[GP1:90,2] + 111.115;
   1:L PR[91] 10mm/sec FINE;
   1:  PR[GP1:91,1] = PR[GP1:90,1] + 95.757;
   1:  PR[GP1:91,2] = PR[GP1:90,2] + 111.000;
   1:L PR[91] 10mm/sec FINE;
   1:  PR[GP1:91,1] = PR[GP1:90,1] + 95.587;
   1:  PR[GP1:91,2] = PR[GP1:90,2] + 111.001;
   1:L PR[91] 10mm/sec FINE;
   1:  PR[GP1:91,1] = PR[GP1:90,1] + 94.768;
   1:  PR[GP1:91,2] = PR[GP1:90,2] + 110.892;
   1:L PR[91] 10mm/sec FINE;
   1:  PR[GP1:91,1] = PR[GP1:90,1] + 93.865;
   1:  PR[GP1:91,2] = PR[GP1:90,2] + 111.244;
   1:L PR[91] 10mm/sec FINE;
   1:  PR[GP1:91,1] = PR[GP1:90,1] + 93.584;
   1:  PR[GP1:91,2] = PR[GP1:90,2] + 111.579;
   1:L PR[91] 10mm/sec FINE;
   1:  PR[GP1:91,1] = PR[GP1:90,1] + 93.241;
   1:  PR[GP1:91,2] = PR[GP1:90,2] + 111.855;
   1:L PR[91] 10mm/sec FINE;
   1:  PR[GP1:91,1] = PR[GP1:90,1] + 93.157;
   1:  PR[GP1:91,2] = PR[GP1:90,2] + 112.025;
   1:L PR[91] 10mm/sec FINE;
   1:  PR[GP1:91,1] = PR[GP1:90,1] + 92.856;
   1:  PR[GP1:91,2] = PR[GP1:90,2] + 112.821;
   1:L PR[91] 10mm/sec FINE;
   1:  PR[GP1:91,1] = PR[GP1:90,1] + 91.959;
   1:  PR[GP1:91,2] = PR[GP1:90,2] + 115.986;
   1:L PR[91] 10mm/sec FINE;
   1:  PR[GP1:91,1] = PR[GP1:90,1] + 91.646;
   1:  PR[GP1:91,2] = PR[GP1:90,2] + 116.658;
   1:L PR[91] 10mm/sec FINE;
   1:  PR[GP1:91,1] = PR[GP1:90,1] + 90.179;
   1:  PR[GP1:91,2] = PR[GP1:90,2] + 119.301;
   1:L PR[91] 10mm/sec FINE;
   1:  PR[GP1:91,1] = PR[GP1:90,1] + 89.931;
   1:  PR[GP1:91,2] = PR[GP1:90,2] + 119.635;
   1:L PR[91] 10mm/sec FINE;
   1:  PR[GP1:91,1] = PR[GP1:90,1] + 87.686;
   1:  PR[GP1:91,2] = PR[GP1:90,2] + 122.205;
   1:L PR[91] 10mm/sec FINE;
   1:  PR[GP1:91,1] = PR[GP1:90,1] + 87.631;
   1:  PR[GP1:91,2] = PR[GP1:90,2] + 122.255;
   1:L PR[91] 10mm/sec FINE;
   1:  PR[GP1:91,1] = PR[GP1:90,1] + 84.763;
   1:  PR[GP1:91,2] = PR[GP1:90,2] + 124.433;
   1:L PR[91] 10mm/sec FINE;
   1:  PR[GP1:91,1] = PR[GP1:90,1] + 81.593;
   1:  PR[GP1:91,2] = PR[GP1:90,2] + 125.940;
   1:L PR[91] 10mm/sec FINE;
   1:  PR[GP1:91,1] = PR[GP1:90,1] + 81.215;
   1:  PR[GP1:91,2] = PR[GP1:90,2] + 126.067;
   1:L PR[91] 10mm/sec FINE;
   1:  PR[GP1:91,1] = PR[GP1:90,1] + 78.295;
   1:  PR[GP1:91,2] = PR[GP1:90,2] + 126.750;
   1:L PR[91] 10mm/sec FINE;
   1:  PR[GP1:91,1] = PR[GP1:90,1] + 77.709;
   1:  PR[GP1:91,2] = PR[GP1:90,2] + 126.844;
   1:L PR[91] 10mm/sec FINE;
   1:  PR[GP1:91,1] = PR[GP1:90,1] + 77.106;
   1:  PR[GP1:91,2] = PR[GP1:90,2] + 126.841;
   1:L PR[91] 10mm/sec FINE;
   1:  PR[GP1:91,1] = PR[GP1:90,1] + 74.219;
   1:  PR[GP1:91,2] = PR[GP1:90,2] + 126.887;
   1:L PR[91] 10mm/sec FINE;
   1:  PR[GP1:91,1] = PR[GP1:90,1] + 73.472;
   1:  PR[GP1:91,2] = PR[GP1:90,2] + 126.759;
   1:L PR[91] 10mm/sec FINE;
   1:  PR[GP1:91,1] = PR[GP1:90,1] + 70.879;
   1:  PR[GP1:91,2] = PR[GP1:90,2] + 126.248;
   1:L PR[91] 10mm/sec FINE;
   1:  PR[GP1:91,1] = PR[GP1:90,1] + 70.041;
   1:  PR[GP1:91,2] = PR[GP1:90,2] + 125.956;
   1:L PR[91] 10mm/sec FINE;
   1:  PR[GP1:91,1] = PR[GP1:90,1] + 67.783;
   1:  PR[GP1:91,2] = PR[GP1:90,2] + 124.986;
   1:L PR[91] 10mm/sec FINE;
   1:  PR[GP1:91,1] = PR[GP1:90,1] + 66.917;
   1:  PR[GP1:91,2] = PR[GP1:90,2] + 124.514;
   1:L PR[91] 10mm/sec FINE;
   1:  PR[GP1:91,1] = PR[GP1:90,1] + 65.021;
   1:  PR[GP1:91,2] = PR[GP1:90,2] + 123.167;
   1:L PR[91] 10mm/sec FINE;
   1:  PR[GP1:91,1] = PR[GP1:90,1] + 64.188;
   1:  PR[GP1:91,2] = PR[GP1:90,2] + 122.514;
   1:L PR[91] 10mm/sec FINE;
   1:  PR[GP1:91,1] = PR[GP1:90,1] + 61.927;
   1:  PR[GP1:91,2] = PR[GP1:90,2] + 120.041;
   1:L PR[91] 10mm/sec FINE;
   1:  PR[GP1:91,1] = PR[GP1:90,1] + 61.323;
   1:  PR[GP1:91,2] = PR[GP1:90,2] + 119.114;
   1:L PR[91] 10mm/sec FINE;
   1:  PR[GP1:91,1] = PR[GP1:90,1] + 60.201;
   1:  PR[GP1:91,2] = PR[GP1:90,2] + 117.194;
   1:L PR[91] 10mm/sec FINE;
   1:  PR[GP1:91,1] = PR[GP1:90,1] + 59.749;
   1:  PR[GP1:91,2] = PR[GP1:90,2] + 116.158;
   1:L PR[91] 10mm/sec FINE;
   1:  PR[GP1:91,1] = PR[GP1:90,1] + 59.059;
   1:  PR[GP1:91,2] = PR[GP1:90,2] + 114.067;
   1:L PR[91] 10mm/sec FINE;
   1:  PR[GP1:91,1] = PR[GP1:90,1] + 58.783;
   1:  PR[GP1:91,2] = PR[GP1:90,2] + 112.972;
   1:L PR[91] 10mm/sec FINE;
   1:  PR[GP1:91,1] = PR[GP1:90,1] + 58.689;
   1:  PR[GP1:91,2] = PR[GP1:90,2] + 111.837;
   1:L PR[91] 10mm/sec FINE;
   1:  PR[GP1:91,1] = PR[GP1:90,1] + 58.459;
   1:  PR[GP1:91,2] = PR[GP1:90,2] + 109.647;
   1:L PR[91] 10mm/sec FINE;
   1:  PR[GP1:91,1] = PR[GP1:90,1] + 58.550;
   1:  PR[GP1:91,2] = PR[GP1:90,2] + 108.542;
   1:L PR[91] 10mm/sec FINE;
   1:  PR[GP1:91,1] = PR[GP1:90,1] + 58.791;
   1:  PR[GP1:91,2] = PR[GP1:90,2] + 106.308;
   1:L PR[91] 10mm/sec FINE;
   1:  PR[GP1:91,1] = PR[GP1:90,1] + 59.052;
   1:  PR[GP1:91,2] = PR[GP1:90,2] + 105.273;
   1:L PR[91] 10mm/sec FINE;
   1:  PR[GP1:91,1] = PR[GP1:90,1] + 59.780;
   1:  PR[GP1:91,2] = PR[GP1:90,2] + 103.065;
   1:L PR[91] 10mm/sec FINE;
   1:  PR[GP1:91,1] = PR[GP1:90,1] + 60.179;
   1:  PR[GP1:91,2] = PR[GP1:90,2] + 102.150;
   1:L PR[91] 10mm/sec FINE;
   1:  PR[GP1:91,1] = PR[GP1:90,1] + 61.425;
   1:  PR[GP1:91,2] = PR[GP1:90,2] + 100.030;
   1:L PR[91] 10mm/sec FINE;
   1:  PR[GP1:91,1] = PR[GP1:90,1] + 61.918;
   1:  PR[GP1:91,2] = PR[GP1:90,2] + 99.273;
   1:L PR[91] 10mm/sec FINE;
   1:  PR[GP1:91,1] = PR[GP1:90,1] + 64.234;
   1:  PR[GP1:91,2] = PR[GP1:90,2] + 96.749;
   1:L PR[91] 10mm/sec FINE;
   1:  PR[GP1:91,1] = PR[GP1:90,1] + 64.846;
   1:  PR[GP1:91,2] = PR[GP1:90,2] + 96.269;
   1:L PR[91] 10mm/sec FINE;
   1:  PR[GP1:91,1] = PR[GP1:90,1] + 67.075;
   1:  PR[GP1:91,2] = PR[GP1:90,2] + 94.694;
   1:L PR[91] 10mm/sec FINE;
   1:  PR[GP1:91,1] = PR[GP1:90,1] + 67.420;
   1:  PR[GP1:91,2] = PR[GP1:90,2] + 94.507;
   1:  PR[GP1:91,3] = PR[GP1:90,3] + 9.900;
   1:L PR[91] 10mm/sec FINE;
   1:  PR[GP1:91,1] = PR[GP1:90,1] + 70.719;
   1:  PR[GP1:91,2] = PR[GP1:90,2] + 93.097;
   1:L PR[91] 10mm/sec FINE;
   1:  PR[GP1:91,1] = PR[GP1:90,1] + 74.252;
   1:  PR[GP1:91,2] = PR[GP1:90,2] + 92.384;
   1:L PR[91] 10mm/sec FINE;
   1:  PR[GP1:91,1] = PR[GP1:90,1] + 74.741;
   1:  PR[GP1:91,2] = PR[GP1:90,2] + 92.356;
   1:L PR[91] 10mm/sec FINE;
   1:  PR[GP1:91,1] = PR[GP1:90,1] + 77.797;
   1:  PR[GP1:91,2] = PR[GP1:90,2] + 92.393;
   1:L PR[91] 10mm/sec FINE;
   1:  PR[GP1:91,1] = PR[GP1:90,1] + 78.686;
   1:  PR[GP1:91,2] = PR[GP1:90,2] + 92.521;
   1:L PR[91] 10mm/sec FINE;
   1:  PR[GP1:91,1] = PR[GP1:90,1] + 81.212;
   1:  PR[GP1:91,2] = PR[GP1:90,2] + 93.091;
   1:L PR[91] 10mm/sec FINE;
   1:  PR[GP1:91,1] = PR[GP1:90,1] + 82.460;
   1:  PR[GP1:91,2] = PR[GP1:90,2] + 93.536;
   1:L PR[91] 10mm/sec FINE;
   1:  PR[GP1:91,1] = PR[GP1:90,1] + 84.372;
   1:  PR[GP1:91,2] = PR[GP1:90,2] + 94.421;
   1:L PR[91] 10mm/sec FINE;
   1:  PR[GP1:91,1] = PR[GP1:90,1] + 85.862;
   1:  PR[GP1:91,2] = PR[GP1:90,2] + 95.322;
   1:L PR[91] 10mm/sec FINE;
   1:  PR[GP1:91,1] = PR[GP1:90,1] + 87.178;
   1:  PR[GP1:91,2] = PR[GP1:90,2] + 96.314;
   1:L PR[91] 10mm/sec FINE;
   1:  PR[GP1:91,1] = PR[GP1:90,1] + 88.730;
   1:  PR[GP1:91,2] = PR[GP1:90,2] + 97.749;
   1:L PR[91] 10mm/sec FINE;
   1:  PR[GP1:91,1] = PR[GP1:90,1] + 89.551;
   1:  PR[GP1:91,2] = PR[GP1:90,2] + 98.705;
   1:L PR[91] 10mm/sec FINE;
   1:  PR[GP1:91,1] = PR[GP1:90,1] + 90.948;
   1:  PR[GP1:91,2] = PR[GP1:90,2] + 100.662;
   1:L PR[91] 10mm/sec FINE;
   1:  PR[GP1:91,1] = PR[GP1:90,1] + 91.421;
   1:  PR[GP1:91,2] = PR[GP1:90,2] + 101.540;
   1:L PR[91] 10mm/sec FINE;
   1:  PR[GP1:91,1] = PR[GP1:90,1] + 92.467;
   1:  PR[GP1:91,2] = PR[GP1:90,2] + 103.888;
   1:L PR[91] 10mm/sec FINE;
   1:  PR[GP1:91,1] = PR[GP1:90,1] + 92.698;
   1:  PR[GP1:91,2] = PR[GP1:90,2] + 104.693;
   1:L PR[91] 10mm/sec FINE;
   1:  PR[GP1:91,1] = PR[GP1:90,1] + 92.742;
   1:  PR[GP1:91,2] = PR[GP1:90,2] + 104.919;
   1:L PR[91] 10mm/sec FINE;
   1:  PR[GP1:91,1] = PR[GP1:90,1] + 92.997;
   1:  PR[GP1:91,2] = PR[GP1:90,2] + 105.583;
   1:L PR[91] 10mm/sec FINE;
   1:  PR[GP1:91,1] = PR[GP1:90,1] + 93.125;
   1:  PR[GP1:91,2] = PR[GP1:90,2] + 105.970;
   1:L PR[91] 10mm/sec FINE;
   1:  PR[GP1:91,1] = PR[GP1:90,1] + 93.306;
   1:  PR[GP1:91,2] = PR[GP1:90,2] + 106.302;
   1:L PR[91] 10mm/sec FINE;
   1:  PR[GP1:91,1] = PR[GP1:90,1] + 93.486;
   1:  PR[GP1:91,2] = PR[GP1:90,2] + 106.444;
   1:L PR[91] 10mm/sec FINE;
   1:  PR[GP1:91,1] = PR[GP1:90,1] + 94.178;
   1:  PR[GP1:91,2] = PR[GP1:90,2] + 107.177;
   1:L PR[91] 10mm/sec FINE;
   1:  PR[GP1:91,1] = PR[GP1:90,1] + 95.293;
   1:  PR[GP1:91,2] = PR[GP1:90,2] + 107.368;
   1:L PR[91] 10mm/sec FINE;
   1:  PR[GP1:91,1] = PR[GP1:90,1] + 96.253;
   1:  PR[GP1:91,2] = PR[GP1:90,2] + 106.712;
   1:L PR[91] 10mm/sec FINE;
   1:  PR[GP1:91,1] = PR[GP1:90,1] + 96.353;
   1:  PR[GP1:91,2] = PR[GP1:90,2] + 106.530;
   1:L PR[91] 10mm/sec FINE;
   1:  PR[GP1:91,1] = PR[GP1:90,1] + 96.553;
   1:  PR[GP1:91,2] = PR[GP1:90,2] + 105.936;
   1:L PR[91] 10mm/sec FINE;
   1:  PR[GP1:91,1] = PR[GP1:90,1] + 96.794;
   1:  PR[GP1:91,2] = PR[GP1:90,2] + 105.339;
   1:L PR[91] 10mm/sec FINE;
   1:  PR[GP1:91,1] = PR[GP1:90,1] + 96.951;
   1:  PR[GP1:91,2] = PR[GP1:90,2] + 104.725;
   1:L PR[91] 10mm/sec FINE;
   1:  PR[GP1:91,1] = PR[GP1:90,1] + 97.246;
   1:  PR[GP1:91,2] = PR[GP1:90,2] + 103.777;
   1:L PR[91] 10mm/sec FINE;
   1:  PR[GP1:91,1] = PR[GP1:90,1] + 98.123;
   1:  PR[GP1:91,2] = PR[GP1:90,2] + 101.831;
   1:L PR[91] 10mm/sec FINE;
   1:  PR[GP1:91,1] = PR[GP1:90,1] + 98.422;
   1:  PR[GP1:91,2] = PR[GP1:90,2] + 101.242;
   1:L PR[91] 10mm/sec FINE;
   1:  PR[GP1:91,1] = PR[GP1:90,1] + 99.767;
   1:  PR[GP1:91,2] = PR[GP1:90,2] + 99.276;
   1:L PR[91] 10mm/sec FINE;
   1:  PR[GP1:91,1] = PR[GP1:90,1] + 99.944;
   1:  PR[GP1:91,2] = PR[GP1:90,2] + 99.036;
   1:L PR[91] 10mm/sec FINE;
   1:  PR[GP1:91,1] = PR[GP1:90,1] + 101.848;
   1:  PR[GP1:91,2] = PR[GP1:90,2] + 97.047;
   1:L PR[91] 10mm/sec FINE;
   1:  PR[GP1:91,1] = PR[GP1:90,1] + 104.119;
   1:  PR[GP1:91,2] = PR[GP1:90,2] + 95.314;
   1:L PR[91] 10mm/sec FINE;
   1:  PR[GP1:91,1] = PR[GP1:90,1] + 106.658;
   1:  PR[GP1:91,2] = PR[GP1:90,2] + 93.950;
   1:L PR[91] 10mm/sec FINE;
   1:  PR[GP1:91,1] = PR[GP1:90,1] + 107.878;
   1:  PR[GP1:91,2] = PR[GP1:90,2] + 93.519;
   1:L PR[91] 10mm/sec FINE;
   1:  PR[GP1:91,1] = PR[GP1:90,1] + 109.354;
   1:  PR[GP1:91,2] = PR[GP1:90,2] + 92.974;
   1:L PR[91] 10mm/sec FINE;
   1:  PR[GP1:91,1] = PR[GP1:90,1] + 112.135;
   1:  PR[GP1:91,2] = PR[GP1:90,2] + 92.405;
   1:L PR[91] 10mm/sec FINE;
   1:  PR[GP1:91,1] = PR[GP1:90,1] + 114.970;
   1:  PR[GP1:91,2] = PR[GP1:90,2] + 92.259;
   1:L PR[91] 10mm/sec FINE;
   1:  PR[GP1:91,1] = PR[GP1:90,1] + 117.743;
   1:  PR[GP1:91,2] = PR[GP1:90,2] + 92.524;
   1:L PR[91] 10mm/sec FINE;
   1:  PR[GP1:91,1] = PR[GP1:90,1] + 120.410;
   1:  PR[GP1:91,2] = PR[GP1:90,2] + 93.196;
   1:L PR[91] 10mm/sec FINE;
   1:  PR[GP1:91,1] = PR[GP1:90,1] + 122.939;
   1:  PR[GP1:91,2] = PR[GP1:90,2] + 94.266;
   1:L PR[91] 10mm/sec FINE;
   1:  PR[GP1:91,1] = PR[GP1:90,1] + 125.270;
   1:  PR[GP1:91,2] = PR[GP1:90,2] + 95.707;
   1:L PR[91] 10mm/sec FINE;
   1:  PR[GP1:91,1] = PR[GP1:90,1] + 127.347;
   1:  PR[GP1:91,2] = PR[GP1:90,2] + 97.485;
   1:L PR[91] 10mm/sec FINE;
   1:  PR[GP1:91,1] = PR[GP1:90,1] + 129.119;
   1:  PR[GP1:91,2] = PR[GP1:90,2] + 99.556;
   1:L PR[91] 10mm/sec FINE;
   1:  PR[GP1:91,1] = PR[GP1:90,1] + 130.545;
   1:  PR[GP1:91,2] = PR[GP1:90,2] + 101.871;
   1:L PR[91] 10mm/sec FINE;
   1:  PR[GP1:91,1] = PR[GP1:90,1] + 131.589;
   1:  PR[GP1:91,2] = PR[GP1:90,2] + 104.374;
   1:L PR[91] 10mm/sec FINE;
   1:  PR[GP1:91,1] = PR[GP1:90,1] + 132.228;
   1:  PR[GP1:91,2] = PR[GP1:90,2] + 107.004;
   1:L PR[91] 10mm/sec FINE;
   1:  PR[GP1:91,1] = PR[GP1:90,1] + 132.448;
   1:  PR[GP1:91,2] = PR[GP1:90,2] + 109.696;
   1:L PR[91] 10mm/sec FINE;
   1:  PR[GP1:91,1] = PR[GP1:90,1] + 132.087;
   1:  PR[GP1:91,2] = PR[GP1:90,2] + 113.097;
   1:L PR[91] 10mm/sec FINE;
   1:  PR[GP1:91,1] = PR[GP1:90,1] + 131.076;
   1:  PR[GP1:91,2] = PR[GP1:90,2] + 116.367;
   1:L PR[91] 10mm/sec FINE;
   1:  PR[GP1:91,1] = PR[GP1:90,1] + 129.432;
   1:  PR[GP1:91,2] = PR[GP1:90,2] + 119.374;
   1:L PR[91] 10mm/sec FINE;
   1:  PR[GP1:91,1] = PR[GP1:90,1] + 127.218;
   1:  PR[GP1:91,2] = PR[GP1:90,2] + 122.003;
   1:L PR[91] 10mm/sec FINE;
   1:  PR[GP1:91,1] = PR[GP1:90,1] + 124.522;
   1:  PR[GP1:91,2] = PR[GP1:90,2] + 124.149;
   1:L PR[91] 10mm/sec FINE;
   1:  PR[GP1:91,1] = PR[GP1:90,1] + 121.450;
   1:  PR[GP1:91,2] = PR[GP1:90,2] + 125.730;
   1:L PR[91] 10mm/sec FINE;
   1:  PR[GP1:91,1] = PR[GP1:90,1] + 118.124;
   1:  PR[GP1:91,2] = PR[GP1:90,2] + 126.684;
   1:L PR[91] 10mm/sec FINE;
   1:  PR[GP1:91,1] = PR[GP1:90,1] + 114.657;
   1:  PR[GP1:91,2] = PR[GP1:90,2] + 126.972;
   1:L PR[91] 10mm/sec FINE;
   1:  PR[GP1:91,1] = PR[GP1:90,1] + 111.162;
   1:  PR[GP1:91,2] = PR[GP1:90,2] + 126.581;
   1:L PR[91] 10mm/sec FINE;
   1:  PR[GP1:91,1] = PR[GP1:90,1] + 107.767;
   1:  PR[GP1:91,2] = PR[GP1:90,2] + 125.524;
   1:L PR[91] 10mm/sec FINE;
   1:  PR[GP1:91,1] = PR[GP1:90,1] + 104.620;
   1:  PR[GP1:91,2] = PR[GP1:90,2] + 123.845;
   1:L PR[91] 10mm/sec FINE;
   1:  PR[GP1:91,1] = PR[GP1:90,1] + 101.823;
   1:  PR[GP1:91,2] = PR[GP1:90,2] + 121.608;
   1:L PR[91] 10mm/sec FINE;
   1:  PR[GP1:91,1] = PR[GP1:90,1] + 99.486;
   1:  PR[GP1:91,2] = PR[GP1:90,2] + 118.893;
   1:L PR[91] 10mm/sec FINE;
   1:  PR[GP1:91,1] = PR[GP1:90,1] + 97.749;
   1:  PR[GP1:91,2] = PR[GP1:90,2] + 115.816;
   1:L PR[91] 10mm/sec FINE;
   1:  PR[GP1:91,1] = PR[GP1:90,1] + 96.891;
   1:  PR[GP1:91,2] = PR[GP1:90,2] + 113.226;
   1:L PR[91] 10mm/sec FINE;
   1:  PR[GP1:91,1] = PR[GP1:90,1] + 96.307;
   1:  PR[GP1:91,2] = PR[GP1:90,2] + 112.161;
   1:L PR[91] 10mm/sec FINE;
   1:  PR[GP1:91,1] = PR[GP1:90,1] + 95.575;
   1:  PR[GP1:91,2] = PR[GP1:90,2] + 111.701;
   1:L PR[91] 10mm/sec FINE;
   1:  PR[GP1:91,1] = PR[GP1:90,1] + 95.221;
   1:  PR[GP1:91,2] = PR[GP1:90,2] + 111.571;
   1:L PR[91] 10mm/sec FINE;
   1:  PR[GP1:91,1] = PR[GP1:90,1] + 94.400;
   1:  PR[GP1:91,2] = PR[GP1:90,2] + 111.692;
   1:L PR[91] 10mm/sec FINE;
   1:  PR[GP1:91,1] = PR[GP1:90,1] + 94.178;
   1:  PR[GP1:91,2] = PR[GP1:90,2] + 111.759;
   1:L PR[91] 10mm/sec FINE;
   1:  PR[GP1:91,1] = PR[GP1:90,1] + 93.258;
   1:  PR[GP1:91,2] = PR[GP1:90,2] + 112.651;
   1:L PR[91] 10mm/sec FINE;
   1:  PR[GP1:91,1] = PR[GP1:90,1] + 92.793;
   1:  PR[GP1:91,2] = PR[GP1:90,2] + 113.744;
   1:L PR[91] 10mm/sec FINE;
   1:  PR[GP1:91,1] = PR[GP1:90,1] + 92.253;
   1:  PR[GP1:91,2] = PR[GP1:90,2] + 115.649;
   1:L PR[91] 10mm/sec FINE;
   1:  PR[GP1:91,1] = PR[GP1:90,1] + 91.545;
   1:  PR[GP1:91,2] = PR[GP1:90,2] + 117.169;
   1:L PR[91] 10mm/sec FINE;
   1:  PR[GP1:91,1] = PR[GP1:90,1] + 90.551;
   1:  PR[GP1:91,2] = PR[GP1:90,2] + 118.961;
   1:L PR[91] 10mm/sec FINE;
   1:  PR[GP1:91,1] = PR[GP1:90,1] + 89.778;
   1:  PR[GP1:91,2] = PR[GP1:90,2] + 120.003;
   1:L PR[91] 10mm/sec FINE;
   1:  PR[GP1:91,1] = PR[GP1:90,1] + 88.127;
   1:  PR[GP1:91,2] = PR[GP1:90,2] + 121.894;
   1:L PR[91] 10mm/sec FINE;
   1:  PR[GP1:91,1] = PR[GP1:90,1] + 87.464;
   1:  PR[GP1:91,2] = PR[GP1:90,2] + 122.493;
   1:L PR[91] 10mm/sec FINE;
   1:  PR[GP1:91,1] = PR[GP1:90,1] + 85.096;
   1:  PR[GP1:91,2] = PR[GP1:90,2] + 124.267;
   1:L PR[91] 10mm/sec FINE;
   1:  PR[GP1:91,1] = PR[GP1:90,1] + 84.659;
   1:  PR[GP1:91,2] = PR[GP1:90,2] + 124.527;
   1:L PR[91] 10mm/sec FINE;
   1:  PR[GP1:91,1] = PR[GP1:90,1] + 81.600;
   1:  PR[GP1:91,2] = PR[GP1:90,2] + 125.946;
   1:L PR[91] 10mm/sec FINE;
   1:  PR[GP1:91,1] = PR[GP1:90,1] + 81.453;
   1:  PR[GP1:91,2] = PR[GP1:90,2] + 125.997;
   1:L PR[91] 10mm/sec FINE;
   1:  PR[GP1:91,1] = PR[GP1:90,1] + 77.900;
   1:  PR[GP1:91,2] = PR[GP1:90,2] + 126.814;
   1:L PR[91] 10mm/sec FINE;
   1:  PR[GP1:91,1] = PR[GP1:90,1] + 74.275;
   1:  PR[GP1:91,2] = PR[GP1:90,2] + 126.870;
   1:L PR[91] 10mm/sec FINE;
   1:  PR[GP1:91,1] = PR[GP1:90,1] + 70.810;
   1:  PR[GP1:91,2] = PR[GP1:90,2] + 126.195;
   1:L PR[91] 10mm/sec FINE;
   1:  PR[GP1:91,1] = PR[GP1:90,1] + 70.396;
   1:  PR[GP1:91,2] = PR[GP1:90,2] + 126.050;
   1:L PR[91] 10mm/sec FINE;
   1:  PR[GP1:91,1] = PR[GP1:90,1] + 67.621;
   1:  PR[GP1:91,2] = PR[GP1:90,2] + 124.858;
   1:L PR[91] 10mm/sec FINE;
   1:  PR[GP1:91,1] = PR[GP1:90,1] + 67.129;
   1:  PR[GP1:91,2] = PR[GP1:90,2] + 124.590;
   1:L PR[91] 10mm/sec FINE;
   1:  PR[GP1:91,1] = PR[GP1:90,1] + 64.799;
   1:  PR[GP1:91,2] = PR[GP1:90,2] + 122.934;
   1:L PR[91] 10mm/sec FINE;
   1:  PR[GP1:91,1] = PR[GP1:90,1] + 64.288;
   1:  PR[GP1:91,2] = PR[GP1:90,2] + 122.534;
   1:L PR[91] 10mm/sec FINE;
   1:  PR[GP1:91,1] = PR[GP1:90,1] + 61.949;
   1:  PR[GP1:91,2] = PR[GP1:90,2] + 119.976;
   1:L PR[91] 10mm/sec FINE;
   1:  PR[GP1:91,1] = PR[GP1:90,1] + 61.563;
   1:  PR[GP1:91,2] = PR[GP1:90,2] + 119.383;
   1:L PR[91] 10mm/sec FINE;
   1:  PR[GP1:91,1] = PR[GP1:90,1] + 60.184;
   1:  PR[GP1:91,2] = PR[GP1:90,2] + 117.024;
   1:L PR[91] 10mm/sec FINE;
   1:  PR[GP1:91,1] = PR[GP1:90,1] + 59.889;
   1:  PR[GP1:91,2] = PR[GP1:90,2] + 116.348;
   1:L PR[91] 10mm/sec FINE;
   1:  PR[GP1:91,1] = PR[GP1:90,1] + 59.041;
   1:  PR[GP1:91,2] = PR[GP1:90,2] + 113.778;
   1:L PR[91] 10mm/sec FINE;
   1:  PR[GP1:91,1] = PR[GP1:90,1] + 58.861;
   1:  PR[GP1:91,2] = PR[GP1:90,2] + 113.063;
   1:L PR[91] 10mm/sec FINE;
   1:  PR[GP1:91,1] = PR[GP1:90,1] + 58.800;
   1:  PR[GP1:91,2] = PR[GP1:90,2] + 112.320;
   1:L PR[91] 10mm/sec FINE;
   1:  PR[GP1:91,1] = PR[GP1:90,1] + 58.516;
   1:  PR[GP1:91,2] = PR[GP1:90,2] + 109.628;
   1:L PR[91] 10mm/sec FINE;
   1:  PR[GP1:91,1] = PR[GP1:90,1] + 58.575;
   1:  PR[GP1:91,2] = PR[GP1:90,2] + 108.920;
   1:L PR[91] 10mm/sec FINE;
   1:  PR[GP1:91,1] = PR[GP1:90,1] + 58.872;
   1:  PR[GP1:91,2] = PR[GP1:90,2] + 106.174;
   1:L PR[91] 10mm/sec FINE;
   1:  PR[GP1:91,1] = PR[GP1:90,1] + 59.033;
   1:  PR[GP1:91,2] = PR[GP1:90,2] + 105.534;
   1:L PR[91] 10mm/sec FINE;
   1:  PR[GP1:91,1] = PR[GP1:90,1] + 59.927;
   1:  PR[GP1:91,2] = PR[GP1:90,2] + 102.820;
   1:L PR[91] 10mm/sec FINE;
   1:  PR[GP1:91,1] = PR[GP1:90,1] + 60.157;
   1:  PR[GP1:91,2] = PR[GP1:90,2] + 102.293;
   1:L PR[91] 10mm/sec FINE;
   1:  PR[GP1:91,1] = PR[GP1:90,1] + 61.688;
   1:  PR[GP1:91,2] = PR[GP1:90,2] + 99.688;
   1:L PR[91] 10mm/sec FINE;
   1:  PR[GP1:91,1] = PR[GP1:90,1] + 61.938;
   1:  PR[GP1:91,2] = PR[GP1:90,2] + 99.304;
   1:L PR[91] 10mm/sec FINE;
   1:  PR[GP1:91,1] = PR[GP1:90,1] + 64.344;
   1:  PR[GP1:91,2] = PR[GP1:90,2] + 96.683;
   1:L PR[91] 10mm/sec FINE;
   1:  PR[GP1:91,1] = PR[GP1:90,1] + 64.584;
   1:  PR[GP1:91,2] = PR[GP1:90,2] + 96.495;
   1:L PR[91] 10mm/sec FINE;
   1:  PR[GP1:91,1] = PR[GP1:90,1] + 67.322;
   1:  PR[GP1:91,2] = PR[GP1:90,2] + 94.560;
   1:L PR[91] 10mm/sec FINE;
   1:  PR[GP1:91,1] = PR[GP1:90,1] + 67.857;
   1:  PR[GP1:91,2] = PR[GP1:90,2] + 94.326;
   1:  PR[GP1:91,3] = PR[GP1:90,3] + 10.900;
   1:L PR[91] 10mm/sec FINE;
   1:  PR[GP1:91,1] = PR[GP1:90,1] + 70.712;
   1:  PR[GP1:91,2] = PR[GP1:90,2] + 93.101;
   1:L PR[91] 10mm/sec FINE;
   1:  PR[GP1:91,1] = PR[GP1:90,1] + 71.549;
   1:  PR[GP1:91,2] = PR[GP1:90,2] + 92.881;
   1:L PR[91] 10mm/sec FINE;
   1:  PR[GP1:91,1] = PR[GP1:90,1] + 74.181;
   1:  PR[GP1:91,2] = PR[GP1:90,2] + 92.356;
   1:L PR[91] 10mm/sec FINE;
   1:  PR[GP1:91,1] = PR[GP1:90,1] + 75.473;
   1:  PR[GP1:91,2] = PR[GP1:90,2] + 92.282;
   1:L PR[91] 10mm/sec FINE;
   1:  PR[GP1:91,1] = PR[GP1:90,1] + 77.665;
   1:  PR[GP1:91,2] = PR[GP1:90,2] + 92.309;
   1:L PR[91] 10mm/sec FINE;
   1:  PR[GP1:91,1] = PR[GP1:90,1] + 79.411;
   1:  PR[GP1:91,2] = PR[GP1:90,2] + 92.559;
   1:L PR[91] 10mm/sec FINE;
   1:  PR[GP1:91,1] = PR[GP1:90,1] + 81.026;
   1:  PR[GP1:91,2] = PR[GP1:90,2] + 92.924;
   1:L PR[91] 10mm/sec FINE;
   1:  PR[GP1:91,1] = PR[GP1:90,1] + 83.149;
   1:  PR[GP1:91,2] = PR[GP1:90,2] + 93.681;
   1:L PR[91] 10mm/sec FINE;
   1:  PR[GP1:91,1] = PR[GP1:90,1] + 84.147;
   1:  PR[GP1:91,2] = PR[GP1:90,2] + 94.143;
   1:L PR[91] 10mm/sec FINE;
   1:  PR[GP1:91,1] = PR[GP1:90,1] + 86.485;
   1:  PR[GP1:91,2] = PR[GP1:90,2] + 95.557;
   1:L PR[91] 10mm/sec FINE;
   1:  PR[GP1:91,1] = PR[GP1:90,1] + 86.942;
   1:  PR[GP1:91,2] = PR[GP1:90,2] + 95.901;
   1:L PR[91] 10mm/sec FINE;
   1:  PR[GP1:91,1] = PR[GP1:90,1] + 89.262;
   1:  PR[GP1:91,2] = PR[GP1:90,2] + 98.048;
   1:L PR[91] 10mm/sec FINE;
   1:  PR[GP1:91,1] = PR[GP1:90,1] + 89.342;
   1:  PR[GP1:91,2] = PR[GP1:90,2] + 98.141;
   1:L PR[91] 10mm/sec FINE;
   1:  PR[GP1:91,1] = PR[GP1:90,1] + 90.259;
   1:  PR[GP1:91,2] = PR[GP1:90,2] + 99.425;
   1:L PR[91] 10mm/sec FINE;
   1:  PR[GP1:91,1] = PR[GP1:90,1] + 91.297;
   1:  PR[GP1:91,2] = PR[GP1:90,2] + 100.841;
   1:L PR[91] 10mm/sec FINE;
   1:  PR[GP1:91,1] = PR[GP1:90,1] + 91.371;
   1:  PR[GP1:91,2] = PR[GP1:90,2] + 100.952;
   1:L PR[91] 10mm/sec FINE;
   1:  PR[GP1:91,1] = PR[GP1:90,1] + 92.674;
   1:  PR[GP1:91,2] = PR[GP1:90,2] + 103.806;
   1:L PR[91] 10mm/sec FINE;
   1:  PR[GP1:91,1] = PR[GP1:90,1] + 92.855;
   1:  PR[GP1:91,2] = PR[GP1:90,2] + 104.354;
   1:L PR[91] 10mm/sec FINE;
   1:  PR[GP1:91,1] = PR[GP1:90,1] + 93.255;
   1:  PR[GP1:91,2] = PR[GP1:90,2] + 105.090;
   1:L PR[91] 10mm/sec FINE;
   1:  PR[GP1:91,1] = PR[GP1:90,1] + 93.663;
   1:  PR[GP1:91,2] = PR[GP1:90,2] + 105.412;
   1:L PR[91] 10mm/sec FINE;
   1:  PR[GP1:91,1] = PR[GP1:90,1] + 94.108;
   1:  PR[GP1:91,2] = PR[GP1:90,2] + 105.883;
   1:L PR[91] 10mm/sec FINE;
   1:  PR[GP1:91,1] = PR[GP1:90,1] + 94.519;
   1:  PR[GP1:91,2] = PR[GP1:90,2] + 105.922;
   1:L PR[91] 10mm/sec FINE;
   1:  PR[GP1:91,1] = PR[GP1:90,1] + 95.164;
   1:  PR[GP1:91,2] = PR[GP1:90,2] + 106.035;
   1:L PR[91] 10mm/sec FINE;
   1:  PR[GP1:91,1] = PR[GP1:90,1] + 96.082;
   1:  PR[GP1:91,2] = PR[GP1:90,2] + 105.423;
   1:L PR[91] 10mm/sec FINE;
   1:  PR[GP1:91,1] = PR[GP1:90,1] + 96.399;
   1:  PR[GP1:91,2] = PR[GP1:90,2] + 104.848;
   1:L PR[91] 10mm/sec FINE;
   1:  PR[GP1:91,1] = PR[GP1:90,1] + 96.810;
   1:  PR[GP1:91,2] = PR[GP1:90,2] + 103.555;
   1:L PR[91] 10mm/sec FINE;
   1:  PR[GP1:91,1] = PR[GP1:90,1] + 97.339;
   1:  PR[GP1:91,2] = PR[GP1:90,2] + 102.357;
   1:L PR[91] 10mm/sec FINE;
   1:  PR[GP1:91,1] = PR[GP1:90,1] + 98.062;
   1:  PR[GP1:91,2] = PR[GP1:90,2] + 100.934;
   1:L PR[91] 10mm/sec FINE;
   1:  PR[GP1:91,1] = PR[GP1:90,1] + 98.841;
   1:  PR[GP1:91,2] = PR[GP1:90,2] + 99.794;
   1:L PR[91] 10mm/sec FINE;
   1:  PR[GP1:91,1] = PR[GP1:90,1] + 99.611;
   1:  PR[GP1:91,2] = PR[GP1:90,2] + 98.756;
   1:L PR[91] 10mm/sec FINE;
   1:  PR[GP1:91,1] = PR[GP1:90,1] + 100.941;
   1:  PR[GP1:91,2] = PR[GP1:90,2] + 97.381;
   1:L PR[91] 10mm/sec FINE;
   1:  PR[GP1:91,1] = PR[GP1:90,1] + 101.496;
   1:  PR[GP1:91,2] = PR[GP1:90,2] + 96.843;
   1:L PR[91] 10mm/sec FINE;
   1:  PR[GP1:91,1] = PR[GP1:90,1] + 103.680;
   1:  PR[GP1:91,2] = PR[GP1:90,2] + 95.226;
   1:L PR[91] 10mm/sec FINE;
   1:  PR[GP1:91,1] = PR[GP1:90,1] + 106.224;
   1:  PR[GP1:91,2] = PR[GP1:90,2] + 93.858;
   1:L PR[91] 10mm/sec FINE;
   1:  PR[GP1:91,1] = PR[GP1:90,1] + 108.974;
   1:  PR[GP1:91,2] = PR[GP1:90,2] + 92.887;
   1:L PR[91] 10mm/sec FINE;
   1:  PR[GP1:91,1] = PR[GP1:90,1] + 111.822;
   1:  PR[GP1:91,2] = PR[GP1:90,2] + 92.329;
   1:L PR[91] 10mm/sec FINE;
   1:  PR[GP1:91,1] = PR[GP1:90,1] + 114.667;
   1:  PR[GP1:91,2] = PR[GP1:90,2] + 92.185;
   1:L PR[91] 10mm/sec FINE;
   1:  PR[GP1:91,1] = PR[GP1:90,1] + 117.497;
   1:  PR[GP1:91,2] = PR[GP1:90,2] + 92.466;
   1:L PR[91] 10mm/sec FINE;
   1:  PR[GP1:91,1] = PR[GP1:90,1] + 120.234;
   1:  PR[GP1:91,2] = PR[GP1:90,2] + 93.158;
   1:L PR[91] 10mm/sec FINE;
   1:  PR[GP1:91,1] = PR[GP1:90,1] + 122.764;
   1:  PR[GP1:91,2] = PR[GP1:90,2] + 94.230;
   1:L PR[91] 10mm/sec FINE;
   1:  PR[GP1:91,1] = PR[GP1:90,1] + 125.096;
   1:  PR[GP1:91,2] = PR[GP1:90,2] + 95.675;
   1:L PR[91] 10mm/sec FINE;
   1:  PR[GP1:91,1] = PR[GP1:90,1] + 127.173;
   1:  PR[GP1:91,2] = PR[GP1:90,2] + 97.456;
   1:L PR[91] 10mm/sec FINE;
   1:  PR[GP1:91,1] = PR[GP1:90,1] + 128.944;
   1:  PR[GP1:91,2] = PR[GP1:90,2] + 99.530;
   1:L PR[91] 10mm/sec FINE;
   1:  PR[GP1:91,1] = PR[GP1:90,1] + 130.369;
   1:  PR[GP1:91,2] = PR[GP1:90,2] + 101.848;
   1:L PR[91] 10mm/sec FINE;
   1:  PR[GP1:91,1] = PR[GP1:90,1] + 131.412;
   1:  PR[GP1:91,2] = PR[GP1:90,2] + 104.353;
   1:L PR[91] 10mm/sec FINE;
   1:  PR[GP1:91,1] = PR[GP1:90,1] + 132.049;
   1:  PR[GP1:91,2] = PR[GP1:90,2] + 106.985;
   1:L PR[91] 10mm/sec FINE;
   1:  PR[GP1:91,1] = PR[GP1:90,1] + 132.208;
   1:  PR[GP1:91,2] = PR[GP1:90,2] + 108.976;
   1:L PR[91] 10mm/sec FINE;
   1:  PR[GP1:91,1] = PR[GP1:90,1] + 132.287;
   1:  PR[GP1:91,2] = PR[GP1:90,2] + 109.683;
   1:L PR[91] 10mm/sec FINE;
   1:  PR[GP1:91,1] = PR[GP1:90,1] + 131.916;
   1:  PR[GP1:91,2] = PR[GP1:90,2] + 113.082;
   1:L PR[91] 10mm/sec FINE;
   1:  PR[GP1:91,1] = PR[GP1:90,1] + 130.902;
   1:  PR[GP1:91,2] = PR[GP1:90,2] + 116.352;
   1:L PR[91] 10mm/sec FINE;
   1:  PR[GP1:91,1] = PR[GP1:90,1] + 129.255;
   1:  PR[GP1:91,2] = PR[GP1:90,2] + 119.360;
   1:L PR[91] 10mm/sec FINE;
   1:  PR[GP1:91,1] = PR[GP1:90,1] + 127.040;
   1:  PR[GP1:91,2] = PR[GP1:90,2] + 121.989;
   1:L PR[91] 10mm/sec FINE;
   1:  PR[GP1:91,1] = PR[GP1:90,1] + 124.343;
   1:  PR[GP1:91,2] = PR[GP1:90,2] + 124.135;
   1:L PR[91] 10mm/sec FINE;
   1:  PR[GP1:91,1] = PR[GP1:90,1] + 121.270;
   1:  PR[GP1:91,2] = PR[GP1:90,2] + 125.715;
   1:L PR[91] 10mm/sec FINE;
   1:  PR[GP1:91,1] = PR[GP1:90,1] + 117.947;
   1:  PR[GP1:91,2] = PR[GP1:90,2] + 126.668;
   1:L PR[91] 10mm/sec FINE;
   1:  PR[GP1:91,1] = PR[GP1:90,1] + 114.416;
   1:  PR[GP1:91,2] = PR[GP1:90,2] + 126.949;
   1:L PR[91] 10mm/sec FINE;
   1:  PR[GP1:91,1] = PR[GP1:90,1] + 110.873;
   1:  PR[GP1:91,2] = PR[GP1:90,2] + 126.552;
   1:L PR[91] 10mm/sec FINE;
   1:  PR[GP1:91,1] = PR[GP1:90,1] + 107.460;
   1:  PR[GP1:91,2] = PR[GP1:90,2] + 125.493;
   1:L PR[91] 10mm/sec FINE;
   1:  PR[GP1:91,1] = PR[GP1:90,1] + 104.248;
   1:  PR[GP1:91,2] = PR[GP1:90,2] + 123.805;
   1:L PR[91] 10mm/sec FINE;
   1:  PR[GP1:91,1] = PR[GP1:90,1] + 101.402;
   1:  PR[GP1:91,2] = PR[GP1:90,2] + 121.557;
   1:L PR[91] 10mm/sec FINE;
   1:  PR[GP1:91,1] = PR[GP1:90,1] + 99.054;
   1:  PR[GP1:91,2] = PR[GP1:90,2] + 118.840;
   1:L PR[91] 10mm/sec FINE;
   1:  PR[GP1:91,1] = PR[GP1:90,1] + 97.282;
   1:  PR[GP1:91,2] = PR[GP1:90,2] + 115.752;
   1:L PR[91] 10mm/sec FINE;
   1:  PR[GP1:91,1] = PR[GP1:90,1] + 96.755;
   1:  PR[GP1:91,2] = PR[GP1:90,2] + 114.163;
   1:L PR[91] 10mm/sec FINE;
   1:  PR[GP1:91,1] = PR[GP1:90,1] + 96.407;
   1:  PR[GP1:91,2] = PR[GP1:90,2] + 113.525;
   1:L PR[91] 10mm/sec FINE;
   1:  PR[GP1:91,1] = PR[GP1:90,1] + 96.129;
   1:  PR[GP1:91,2] = PR[GP1:90,2] + 113.114;
   1:L PR[91] 10mm/sec FINE;
   1:  PR[GP1:91,1] = PR[GP1:90,1] + 95.449;
   1:  PR[GP1:91,2] = PR[GP1:90,2] + 112.717;
   1:L PR[91] 10mm/sec FINE;
   1:  PR[GP1:91,1] = PR[GP1:90,1] + 95.113;
   1:  PR[GP1:91,2] = PR[GP1:90,2] + 112.585;
   1:L PR[91] 10mm/sec FINE;
   1:  PR[GP1:91,1] = PR[GP1:90,1] + 94.725;
   1:  PR[GP1:91,2] = PR[GP1:90,2] + 112.734;
   1:L PR[91] 10mm/sec FINE;
   1:  PR[GP1:91,1] = PR[GP1:90,1] + 94.013;
   1:  PR[GP1:91,2] = PR[GP1:90,2] + 112.847;
   1:L PR[91] 10mm/sec FINE;
   1:  PR[GP1:91,1] = PR[GP1:90,1] + 93.537;
   1:  PR[GP1:91,2] = PR[GP1:90,2] + 113.402;
   1:L PR[91] 10mm/sec FINE;
   1:  PR[GP1:91,1] = PR[GP1:90,1] + 93.088;
   1:  PR[GP1:91,2] = PR[GP1:90,2] + 113.838;
   1:L PR[91] 10mm/sec FINE;
   1:  PR[GP1:91,1] = PR[GP1:90,1] + 92.728;
   1:  PR[GP1:91,2] = PR[GP1:90,2] + 114.672;
   1:L PR[91] 10mm/sec FINE;
   1:  PR[GP1:91,1] = PR[GP1:90,1] + 92.547;
   1:  PR[GP1:91,2] = PR[GP1:90,2] + 115.312;
   1:L PR[91] 10mm/sec FINE;
   1:  PR[GP1:91,1] = PR[GP1:90,1] + 91.445;
   1:  PR[GP1:91,2] = PR[GP1:90,2] + 117.680;
   1:L PR[91] 10mm/sec FINE;
   1:  PR[GP1:91,1] = PR[GP1:90,1] + 90.922;
   1:  PR[GP1:91,2] = PR[GP1:90,2] + 118.621;
   1:L PR[91] 10mm/sec FINE;
   1:  PR[GP1:91,1] = PR[GP1:90,1] + 89.626;
   1:  PR[GP1:91,2] = PR[GP1:90,2] + 120.371;
   1:L PR[91] 10mm/sec FINE;
   1:  PR[GP1:91,1] = PR[GP1:90,1] + 88.567;
   1:  PR[GP1:91,2] = PR[GP1:90,2] + 121.583;
   1:L PR[91] 10mm/sec FINE;
   1:  PR[GP1:91,1] = PR[GP1:90,1] + 87.296;
   1:  PR[GP1:91,2] = PR[GP1:90,2] + 122.731;
   1:L PR[91] 10mm/sec FINE;
   1:  PR[GP1:91,1] = PR[GP1:90,1] + 85.595;
   1:  PR[GP1:91,2] = PR[GP1:90,2] + 124.005;
   1:L PR[91] 10mm/sec FINE;
   1:  PR[GP1:91,1] = PR[GP1:90,1] + 84.503;
   1:  PR[GP1:91,2] = PR[GP1:90,2] + 124.654;
   1:L PR[91] 10mm/sec FINE;
   1:  PR[GP1:91,1] = PR[GP1:90,1] + 82.144;
   1:  PR[GP1:91,2] = PR[GP1:90,2] + 125.749;
   1:L PR[91] 10mm/sec FINE;
   1:  PR[GP1:91,1] = PR[GP1:90,1] + 81.327;
   1:  PR[GP1:91,2] = PR[GP1:90,2] + 126.036;
   1:L PR[91] 10mm/sec FINE;
   1:  PR[GP1:91,1] = PR[GP1:90,1] + 78.385;
   1:  PR[GP1:91,2] = PR[GP1:90,2] + 126.712;
   1:L PR[91] 10mm/sec FINE;
   1:  PR[GP1:91,1] = PR[GP1:90,1] + 77.880;
   1:  PR[GP1:91,2] = PR[GP1:90,2] + 126.784;
   1:L PR[91] 10mm/sec FINE;
   1:  PR[GP1:91,1] = PR[GP1:90,1] + 74.511;
   1:  PR[GP1:91,2] = PR[GP1:90,2] + 126.843;
   1:L PR[91] 10mm/sec FINE;
   1:  PR[GP1:91,1] = PR[GP1:90,1] + 74.302;
   1:  PR[GP1:91,2] = PR[GP1:90,2] + 126.831;
   1:L PR[91] 10mm/sec FINE;
   1:  PR[GP1:91,1] = PR[GP1:90,1] + 70.748;
   1:  PR[GP1:91,2] = PR[GP1:90,2] + 126.143;
   1:L PR[91] 10mm/sec FINE;
   1:  PR[GP1:91,1] = PR[GP1:90,1] + 67.459;
   1:  PR[GP1:91,2] = PR[GP1:90,2] + 124.730;
   1:L PR[91] 10mm/sec FINE;
   1:  PR[GP1:91,1] = PR[GP1:90,1] + 67.341;
   1:  PR[GP1:91,2] = PR[GP1:90,2] + 124.666;
   1:L PR[91] 10mm/sec FINE;
   1:  PR[GP1:91,1] = PR[GP1:90,1] + 64.577;
   1:  PR[GP1:91,2] = PR[GP1:90,2] + 122.702;
   1:L PR[91] 10mm/sec FINE;
   1:  PR[GP1:91,1] = PR[GP1:90,1] + 64.388;
   1:  PR[GP1:91,2] = PR[GP1:90,2] + 122.554;
   1:L PR[91] 10mm/sec FINE;
   1:  PR[GP1:91,1] = PR[GP1:90,1] + 61.972;
   1:  PR[GP1:91,2] = PR[GP1:90,2] + 119.912;
   1:L PR[91] 10mm/sec FINE;
   1:  PR[GP1:91,1] = PR[GP1:90,1] + 61.803;
   1:  PR[GP1:91,2] = PR[GP1:90,2] + 119.652;
   1:L PR[91] 10mm/sec FINE;
   1:  PR[GP1:91,1] = PR[GP1:90,1] + 60.167;
   1:  PR[GP1:91,2] = PR[GP1:90,2] + 116.853;
   1:L PR[91] 10mm/sec FINE;
   1:  PR[GP1:91,1] = PR[GP1:90,1] + 60.029;
   1:  PR[GP1:91,2] = PR[GP1:90,2] + 116.538;
   1:L PR[91] 10mm/sec FINE;
   1:  PR[GP1:91,1] = PR[GP1:90,1] + 59.024;
   1:  PR[GP1:91,2] = PR[GP1:90,2] + 113.489;
   1:L PR[91] 10mm/sec FINE;
   1:  PR[GP1:91,1] = PR[GP1:90,1] + 58.939;
   1:  PR[GP1:91,2] = PR[GP1:90,2] + 113.153;
   1:L PR[91] 10mm/sec FINE;
   1:  PR[GP1:91,1] = PR[GP1:90,1] + 58.574;
   1:  PR[GP1:91,2] = PR[GP1:90,2] + 109.612;
   1:L PR[91] 10mm/sec FINE;
   1:  PR[GP1:91,1] = PR[GP1:90,1] + 58.952;
   1:  PR[GP1:91,2] = PR[GP1:90,2] + 106.040;
   1:L PR[91] 10mm/sec FINE;
   1:  PR[GP1:91,1] = PR[GP1:90,1] + 59.014;
   1:  PR[GP1:91,2] = PR[GP1:90,2] + 105.795;
   1:L PR[91] 10mm/sec FINE;
   1:  PR[GP1:91,1] = PR[GP1:90,1] + 60.074;
   1:  PR[GP1:91,2] = PR[GP1:90,2] + 102.575;
   1:L PR[91] 10mm/sec FINE;
   1:  PR[GP1:91,1] = PR[GP1:90,1] + 60.135;
   1:  PR[GP1:91,2] = PR[GP1:90,2] + 102.436;
   1:L PR[91] 10mm/sec FINE;
   1:  PR[GP1:91,1] = PR[GP1:90,1] + 61.943;
   1:  PR[GP1:91,2] = PR[GP1:90,2] + 99.360;
   1:L PR[91] 10mm/sec FINE;
   1:  PR[GP1:91,1] = PR[GP1:90,1] + 64.447;
   1:  PR[GP1:91,2] = PR[GP1:90,2] + 96.644;
   1:L PR[91] 10mm/sec FINE;
   1:  PR[GP1:91,1] = PR[GP1:90,1] + 64.590;
   1:  PR[GP1:91,2] = PR[GP1:90,2] + 96.534;
   1:L PR[91] 10mm/sec FINE;
   1:  PR[GP1:91,1] = PR[GP1:90,1] + 67.415;
   1:  PR[GP1:91,2] = PR[GP1:90,2] + 94.543;
   1:L PR[91] 10mm/sec FINE;
   1:  PR[GP1:91,1] = PR[GP1:90,1] + 68.523;
   1:  PR[GP1:91,2] = PR[GP1:90,2] + 94.041;
   1:  PR[GP1:91,3] = PR[GP1:90,3] + 11.900;
   1:L PR[91] 10mm/sec FINE;
   1:  PR[GP1:91,1] = PR[GP1:90,1] + 70.700;
   1:  PR[GP1:91,2] = PR[GP1:90,2] + 93.107;
   1:L PR[91] 10mm/sec FINE;
   1:  PR[GP1:91,1] = PR[GP1:90,1] + 72.260;
   1:  PR[GP1:91,2] = PR[GP1:90,2] + 92.697;
   1:L PR[91] 10mm/sec FINE;
   1:  PR[GP1:91,1] = PR[GP1:90,1] + 74.109;
   1:  PR[GP1:91,2] = PR[GP1:90,2] + 92.328;
   1:L PR[91] 10mm/sec FINE;
   1:  PR[GP1:91,1] = PR[GP1:90,1] + 76.204;
   1:  PR[GP1:91,2] = PR[GP1:90,2] + 92.208;
   1:L PR[91] 10mm/sec FINE;
   1:  PR[GP1:91,1] = PR[GP1:90,1] + 77.533;
   1:  PR[GP1:91,2] = PR[GP1:90,2] + 92.224;
   1:L PR[91] 10mm/sec FINE;
   1:  PR[GP1:91,1] = PR[GP1:90,1] + 80.137;
   1:  PR[GP1:91,2] = PR[GP1:90,2] + 92.598;
   1:L PR[91] 10mm/sec FINE;
   1:  PR[GP1:91,1] = PR[GP1:90,1] + 80.840;
   1:  PR[GP1:91,2] = PR[GP1:90,2] + 92.756;
   1:L PR[91] 10mm/sec FINE;
   1:  PR[GP1:91,1] = PR[GP1:90,1] + 83.837;
   1:  PR[GP1:91,2] = PR[GP1:90,2] + 93.826;
   1:L PR[91] 10mm/sec FINE;
   1:  PR[GP1:91,1] = PR[GP1:90,1] + 83.923;
   1:  PR[GP1:91,2] = PR[GP1:90,2] + 93.866;
   1:L PR[91] 10mm/sec FINE;
   1:  PR[GP1:91,1] = PR[GP1:90,1] + 84.487;
   1:  PR[GP1:91,2] = PR[GP1:90,2] + 94.207;
   1:L PR[91] 10mm/sec FINE;
   1:  PR[GP1:91,1] = PR[GP1:90,1] + 86.697;
   1:  PR[GP1:91,2] = PR[GP1:90,2] + 95.479;
   1:L PR[91] 10mm/sec FINE;
   1:  PR[GP1:91,1] = PR[GP1:90,1] + 87.040;
   1:  PR[GP1:91,2] = PR[GP1:90,2] + 95.697;
   1:L PR[91] 10mm/sec FINE;
   1:  PR[GP1:91,1] = PR[GP1:90,1] + 89.112;
   1:  PR[GP1:91,2] = PR[GP1:90,2] + 97.542;
   1:L PR[91] 10mm/sec FINE;
   1:  PR[GP1:91,1] = PR[GP1:90,1] + 89.741;
   1:  PR[GP1:91,2] = PR[GP1:90,2] + 98.159;
   1:L PR[91] 10mm/sec FINE;
   1:  PR[GP1:91,1] = PR[GP1:90,1] + 91.136;
   1:  PR[GP1:91,2] = PR[GP1:90,2] + 100.061;
   1:L PR[91] 10mm/sec FINE;
   1:  PR[GP1:91,1] = PR[GP1:90,1] + 91.812;
   1:  PR[GP1:91,2] = PR[GP1:90,2] + 101.086;
   1:L PR[91] 10mm/sec FINE;
   1:  PR[GP1:91,1] = PR[GP1:90,1] + 92.646;
   1:  PR[GP1:91,2] = PR[GP1:90,2] + 102.908;
   1:L PR[91] 10mm/sec FINE;
   1:  PR[GP1:91,1] = PR[GP1:90,1] + 92.865;
   1:  PR[GP1:91,2] = PR[GP1:90,2] + 103.253;
   1:L PR[91] 10mm/sec FINE;
   1:  PR[GP1:91,1] = PR[GP1:90,1] + 93.204;
   1:  PR[GP1:91,2] = PR[GP1:90,2] + 103.878;
   1:L PR[91] 10mm/sec FINE;
   1:  PR[GP1:91,1] = PR[GP1:90,1] + 93.841;
   1:  PR[GP1:91,2] = PR[GP1:90,2] + 104.379;
   1:L PR[91] 10mm/sec FINE;
   1:  PR[GP1:91,1] = PR[GP1:90,1] + 94.033;
   1:  PR[GP1:91,2] = PR[GP1:90,2] + 104.583;
   1:L PR[91] 10mm/sec FINE;
   1:  PR[GP1:91,1] = PR[GP1:90,1] + 94.736;
   1:  PR[GP1:91,2] = PR[GP1:90,2] + 104.650;
   1:L PR[91] 10mm/sec FINE;
   1:  PR[GP1:91,1] = PR[GP1:90,1] + 95.035;
   1:  PR[GP1:91,2] = PR[GP1:90,2] + 104.703;
   1:L PR[91] 10mm/sec FINE;
   1:  PR[GP1:91,1] = PR[GP1:90,1] + 95.912;
   1:  PR[GP1:91,2] = PR[GP1:90,2] + 104.134;
   1:L PR[91] 10mm/sec FINE;
   1:  PR[GP1:91,1] = PR[GP1:90,1] + 96.442;
   1:  PR[GP1:91,2] = PR[GP1:90,2] + 103.173;
   1:L PR[91] 10mm/sec FINE;
   1:  PR[GP1:91,1] = PR[GP1:90,1] + 96.558;
   1:  PR[GP1:91,2] = PR[GP1:90,2] + 102.880;
   1:L PR[91] 10mm/sec FINE;
   1:  PR[GP1:91,1] = PR[GP1:90,1] + 97.702;
   1:  PR[GP1:91,2] = PR[GP1:90,2] + 100.625;
   1:L PR[91] 10mm/sec FINE;
   1:  PR[GP1:91,1] = PR[GP1:90,1] + 97.916;
   1:  PR[GP1:91,2] = PR[GP1:90,2] + 100.313;
   1:L PR[91] 10mm/sec FINE;
   1:  PR[GP1:91,1] = PR[GP1:90,1] + 99.278;
   1:  PR[GP1:91,2] = PR[GP1:90,2] + 98.476;
   1:L PR[91] 10mm/sec FINE;
   1:  PR[GP1:91,1] = PR[GP1:90,1] + 99.871;
   1:  PR[GP1:91,2] = PR[GP1:90,2] + 97.863;
   1:L PR[91] 10mm/sec FINE;
   1:  PR[GP1:91,1] = PR[GP1:90,1] + 101.183;
   1:  PR[GP1:91,2] = PR[GP1:90,2] + 96.593;
   1:L PR[91] 10mm/sec FINE;
   1:  PR[GP1:91,1] = PR[GP1:90,1] + 102.440;
   1:  PR[GP1:91,2] = PR[GP1:90,2] + 95.660;
   1:L PR[91] 10mm/sec FINE;
   1:  PR[GP1:91,1] = PR[GP1:90,1] + 103.376;
   1:  PR[GP1:91,2] = PR[GP1:90,2] + 95.007;
   1:L PR[91] 10mm/sec FINE;
   1:  PR[GP1:91,1] = PR[GP1:90,1] + 105.817;
   1:  PR[GP1:91,2] = PR[GP1:90,2] + 93.746;
   1:L PR[91] 10mm/sec FINE;
   1:  PR[GP1:91,1] = PR[GP1:90,1] + 108.551;
   1:  PR[GP1:91,2] = PR[GP1:90,2] + 92.789;
   1:L PR[91] 10mm/sec FINE;
   1:  PR[GP1:91,1] = PR[GP1:90,1] + 111.441;
   1:  PR[GP1:91,2] = PR[GP1:90,2] + 92.237;
   1:L PR[91] 10mm/sec FINE;
   1:  PR[GP1:91,1] = PR[GP1:90,1] + 114.363;
   1:  PR[GP1:91,2] = PR[GP1:90,2] + 92.111;
   1:L PR[91] 10mm/sec FINE;
   1:  PR[GP1:91,1] = PR[GP1:90,1] + 117.201;
   1:  PR[GP1:91,2] = PR[GP1:90,2] + 92.394;
   1:L PR[91] 10mm/sec FINE;
   1:  PR[GP1:91,1] = PR[GP1:90,1] + 119.956;
   1:  PR[GP1:91,2] = PR[GP1:90,2] + 93.093;
   1:L PR[91] 10mm/sec FINE;
   1:  PR[GP1:91,1] = PR[GP1:90,1] + 122.564;
   1:  PR[GP1:91,2] = PR[GP1:90,2] + 94.189;
   1:L PR[91] 10mm/sec FINE;
   1:  PR[GP1:91,1] = PR[GP1:90,1] + 123.469;
   1:  PR[GP1:91,2] = PR[GP1:90,2] + 94.741;
   1:L PR[91] 10mm/sec FINE;
   1:  PR[GP1:91,1] = PR[GP1:90,1] + 124.922;
   1:  PR[GP1:91,2] = PR[GP1:90,2] + 95.643;
   1:L PR[91] 10mm/sec FINE;
   1:  PR[GP1:91,1] = PR[GP1:90,1] + 126.998;
   1:  PR[GP1:91,2] = PR[GP1:90,2] + 97.427;
   1:L PR[91] 10mm/sec FINE;
   1:  PR[GP1:91,1] = PR[GP1:90,1] + 128.770;
   1:  PR[GP1:91,2] = PR[GP1:90,2] + 99.504;
   1:L PR[91] 10mm/sec FINE;
   1:  PR[GP1:91,1] = PR[GP1:90,1] + 130.193;
   1:  PR[GP1:91,2] = PR[GP1:90,2] + 101.825;
   1:L PR[91] 10mm/sec FINE;
   1:  PR[GP1:91,1] = PR[GP1:90,1] + 131.235;
   1:  PR[GP1:91,2] = PR[GP1:90,2] + 104.332;
   1:L PR[91] 10mm/sec FINE;
   1:  PR[GP1:91,1] = PR[GP1:90,1] + 131.870;
   1:  PR[GP1:91,2] = PR[GP1:90,2] + 106.966;
   1:L PR[91] 10mm/sec FINE;
   1:  PR[GP1:91,1] = PR[GP1:90,1] + 131.984;
   1:  PR[GP1:91,2] = PR[GP1:90,2] + 108.389;
   1:L PR[91] 10mm/sec FINE;
   1:  PR[GP1:91,1] = PR[GP1:90,1] + 132.125;
   1:  PR[GP1:91,2] = PR[GP1:90,2] + 109.667;
   1:L PR[91] 10mm/sec FINE;
   1:  PR[GP1:91,1] = PR[GP1:90,1] + 131.914;
   1:  PR[GP1:91,2] = PR[GP1:90,2] + 111.457;
   1:L PR[91] 10mm/sec FINE;
   1:  PR[GP1:91,1] = PR[GP1:90,1] + 131.745;
   1:  PR[GP1:91,2] = PR[GP1:90,2] + 113.067;
   1:L PR[91] 10mm/sec FINE;
   1:  PR[GP1:91,1] = PR[GP1:90,1] + 130.728;
   1:  PR[GP1:91,2] = PR[GP1:90,2] + 116.338;
   1:L PR[91] 10mm/sec FINE;
   1:  PR[GP1:91,1] = PR[GP1:90,1] + 129.078;
   1:  PR[GP1:91,2] = PR[GP1:90,2] + 119.346;
   1:L PR[91] 10mm/sec FINE;
   1:  PR[GP1:91,1] = PR[GP1:90,1] + 126.861;
   1:  PR[GP1:91,2] = PR[GP1:90,2] + 121.975;
   1:L PR[91] 10mm/sec FINE;
   1:  PR[GP1:91,1] = PR[GP1:90,1] + 124.163;
   1:  PR[GP1:91,2] = PR[GP1:90,2] + 124.120;
   1:L PR[91] 10mm/sec FINE;
   1:  PR[GP1:91,1] = PR[GP1:90,1] + 121.406;
   1:  PR[GP1:91,2] = PR[GP1:90,2] + 125.538;
   1:L PR[91] 10mm/sec FINE;
   1:  PR[GP1:91,1] = PR[GP1:90,1] + 121.083;
   1:  PR[GP1:91,2] = PR[GP1:90,2] + 125.699;
   1:L PR[91] 10mm/sec FINE;
   1:  PR[GP1:91,1] = PR[GP1:90,1] + 117.666;
   1:  PR[GP1:91,2] = PR[GP1:90,2] + 126.643;
   1:L PR[91] 10mm/sec FINE;
   1:  PR[GP1:91,1] = PR[GP1:90,1] + 114.118;
   1:  PR[GP1:91,2] = PR[GP1:90,2] + 126.921;
   1:L PR[91] 10mm/sec FINE;
   1:  PR[GP1:91,1] = PR[GP1:90,1] + 110.572;
   1:  PR[GP1:91,2] = PR[GP1:90,2] + 126.522;
   1:L PR[91] 10mm/sec FINE;
   1:  PR[GP1:91,1] = PR[GP1:90,1] + 107.078;
   1:  PR[GP1:91,2] = PR[GP1:90,2] + 125.451;
   1:L PR[91] 10mm/sec FINE;
   1:  PR[GP1:91,1] = PR[GP1:90,1] + 103.842;
   1:  PR[GP1:91,2] = PR[GP1:90,2] + 123.757;
   1:L PR[91] 10mm/sec FINE;
   1:  PR[GP1:91,1] = PR[GP1:90,1] + 100.970;
   1:  PR[GP1:91,2] = PR[GP1:90,2] + 121.504;
   1:L PR[91] 10mm/sec FINE;
   1:  PR[GP1:91,1] = PR[GP1:90,1] + 98.589;
   1:  PR[GP1:91,2] = PR[GP1:90,2] + 118.773;
   1:L PR[91] 10mm/sec FINE;
   1:  PR[GP1:91,1] = PR[GP1:90,1] + 96.814;
   1:  PR[GP1:91,2] = PR[GP1:90,2] + 115.688;
   1:L PR[91] 10mm/sec FINE;
   1:  PR[GP1:91,1] = PR[GP1:90,1] + 96.619;
   1:  PR[GP1:91,2] = PR[GP1:90,2] + 115.099;
   1:L PR[91] 10mm/sec FINE;
   1:  PR[GP1:91,1] = PR[GP1:90,1] + 96.481;
   1:  PR[GP1:91,2] = PR[GP1:90,2] + 114.847;
   1:L PR[91] 10mm/sec FINE;
   1:  PR[GP1:91,1] = PR[GP1:90,1] + 95.961;
   1:  PR[GP1:91,2] = PR[GP1:90,2] + 114.075;
   1:L PR[91] 10mm/sec FINE;
   1:  PR[GP1:91,1] = PR[GP1:90,1] + 95.589;
   1:  PR[GP1:91,2] = PR[GP1:90,2] + 113.859;
   1:L PR[91] 10mm/sec FINE;
   1:  PR[GP1:91,1] = PR[GP1:90,1] + 94.926;
   1:  PR[GP1:91,2] = PR[GP1:90,2] + 113.597;
   1:L PR[91] 10mm/sec FINE;
   1:  PR[GP1:91,1] = PR[GP1:90,1] + 94.095;
   1:  PR[GP1:91,2] = PR[GP1:90,2] + 113.916;
   1:L PR[91] 10mm/sec FINE;
   1:  PR[GP1:91,1] = PR[GP1:90,1] + 93.821;
   1:  PR[GP1:91,2] = PR[GP1:90,2] + 113.960;
   1:L PR[91] 10mm/sec FINE;
   1:  PR[GP1:91,1] = PR[GP1:90,1] + 93.139;
   1:  PR[GP1:91,2] = PR[GP1:90,2] + 114.754;
   1:L PR[91] 10mm/sec FINE;
   1:  PR[GP1:91,1] = PR[GP1:90,1] + 92.932;
   1:  PR[GP1:91,2] = PR[GP1:90,2] + 114.957;
   1:L PR[91] 10mm/sec FINE;
   1:  PR[GP1:91,1] = PR[GP1:90,1] + 91.291;
   1:  PR[GP1:91,2] = PR[GP1:90,2] + 118.285;
   1:L PR[91] 10mm/sec FINE;
   1:  PR[GP1:91,1] = PR[GP1:90,1] + 89.473;
   1:  PR[GP1:91,2] = PR[GP1:90,2] + 120.739;
   1:L PR[91] 10mm/sec FINE;
   1:  PR[GP1:91,1] = PR[GP1:90,1] + 89.007;
   1:  PR[GP1:91,2] = PR[GP1:90,2] + 121.272;
   1:L PR[91] 10mm/sec FINE;
   1:  PR[GP1:91,1] = PR[GP1:90,1] + 87.128;
   1:  PR[GP1:91,2] = PR[GP1:90,2] + 122.969;
   1:L PR[91] 10mm/sec FINE;
   1:  PR[GP1:91,1] = PR[GP1:90,1] + 86.094;
   1:  PR[GP1:91,2] = PR[GP1:90,2] + 123.744;
   1:L PR[91] 10mm/sec FINE;
   1:  PR[GP1:91,1] = PR[GP1:90,1] + 84.347;
   1:  PR[GP1:91,2] = PR[GP1:90,2] + 124.782;
   1:L PR[91] 10mm/sec FINE;
   1:  PR[GP1:91,1] = PR[GP1:90,1] + 82.688;
   1:  PR[GP1:91,2] = PR[GP1:90,2] + 125.551;
   1:L PR[91] 10mm/sec FINE;
   1:  PR[GP1:91,1] = PR[GP1:90,1] + 81.200;
   1:  PR[GP1:91,2] = PR[GP1:90,2] + 126.074;
   1:L PR[91] 10mm/sec FINE;
   1:  PR[GP1:91,1] = PR[GP1:90,1] + 78.957;
   1:  PR[GP1:91,2] = PR[GP1:90,2] + 126.590;
   1:L PR[91] 10mm/sec FINE;
   1:  PR[GP1:91,1] = PR[GP1:90,1] + 77.794;
   1:  PR[GP1:91,2] = PR[GP1:90,2] + 126.754;
   1:L PR[91] 10mm/sec FINE;
   1:  PR[GP1:91,1] = PR[GP1:90,1] + 75.093;
   1:  PR[GP1:91,2] = PR[GP1:90,2] + 126.802;
   1:L PR[91] 10mm/sec FINE;
   1:  PR[GP1:91,1] = PR[GP1:90,1] + 74.263;
   1:  PR[GP1:91,2] = PR[GP1:90,2] + 126.753;
   1:L PR[91] 10mm/sec FINE;
   1:  PR[GP1:91,1] = PR[GP1:90,1] + 71.293;
   1:  PR[GP1:91,2] = PR[GP1:90,2] + 126.178;
   1:L PR[91] 10mm/sec FINE;
   1:  PR[GP1:91,1] = PR[GP1:90,1] + 70.761;
   1:  PR[GP1:91,2] = PR[GP1:90,2] + 126.038;
   1:L PR[91] 10mm/sec FINE;
   1:  PR[GP1:91,1] = PR[GP1:90,1] + 67.745;
   1:  PR[GP1:91,2] = PR[GP1:90,2] + 124.759;
   1:L PR[91] 10mm/sec FINE;
   1:  PR[GP1:91,1] = PR[GP1:90,1] + 67.448;
   1:  PR[GP1:91,2] = PR[GP1:90,2] + 124.612;
   1:L PR[91] 10mm/sec FINE;
   1:  PR[GP1:91,1] = PR[GP1:90,1] + 64.619;
   1:  PR[GP1:91,2] = PR[GP1:90,2] + 122.625;
   1:L PR[91] 10mm/sec FINE;
   1:  PR[GP1:91,1] = PR[GP1:90,1] + 64.485;
   1:  PR[GP1:91,2] = PR[GP1:90,2] + 122.521;
   1:L PR[91] 10mm/sec FINE;
   1:  PR[GP1:91,1] = PR[GP1:90,1] + 62.015;
   1:  PR[GP1:91,2] = PR[GP1:90,2] + 119.841;
   1:L PR[91] 10mm/sec FINE;
   1:  PR[GP1:91,1] = PR[GP1:90,1] + 60.166;
   1:  PR[GP1:91,2] = PR[GP1:90,2] + 116.696;
   1:L PR[91] 10mm/sec FINE;
   1:  PR[GP1:91,1] = PR[GP1:90,1] + 59.022;
   1:  PR[GP1:91,2] = PR[GP1:90,2] + 113.227;
   1:L PR[91] 10mm/sec FINE;
   1:  PR[GP1:91,1] = PR[GP1:90,1] + 58.646;
   1:  PR[GP1:91,2] = PR[GP1:90,2] + 109.589;
   1:L PR[91] 10mm/sec FINE;
   1:  PR[GP1:91,1] = PR[GP1:90,1] + 59.061;
   1:  PR[GP1:91,2] = PR[GP1:90,2] + 105.947;
   1:L PR[91] 10mm/sec FINE;
   1:  PR[GP1:91,1] = PR[GP1:90,1] + 60.222;
   1:  PR[GP1:91,2] = PR[GP1:90,2] + 102.480;
   1:L PR[91] 10mm/sec FINE;
   1:  PR[GP1:91,1] = PR[GP1:90,1] + 60.377;
   1:  PR[GP1:91,2] = PR[GP1:90,2] + 102.205;
   1:L PR[91] 10mm/sec FINE;
   1:  PR[GP1:91,1] = PR[GP1:90,1] + 62.082;
   1:  PR[GP1:91,2] = PR[GP1:90,2] + 99.340;
   1:L PR[91] 10mm/sec FINE;
   1:  PR[GP1:91,1] = PR[GP1:90,1] + 62.434;
   1:  PR[GP1:91,2] = PR[GP1:90,2] + 98.934;
   1:L PR[91] 10mm/sec FINE;
   1:  PR[GP1:91,1] = PR[GP1:90,1] + 64.537;
   1:  PR[GP1:91,2] = PR[GP1:90,2] + 96.665;
   1:L PR[91] 10mm/sec FINE;
   1:  PR[GP1:91,1] = PR[GP1:90,1] + 65.192;
   1:  PR[GP1:91,2] = PR[GP1:90,2] + 96.160;
   1:L PR[91] 10mm/sec FINE;
   1:  PR[GP1:91,1] = PR[GP1:90,1] + 67.458;
   1:  PR[GP1:91,2] = PR[GP1:90,2] + 94.563;
   1:L PR[91] 10mm/sec FINE;
   1:  PR[GP1:91,1] = PR[GP1:90,1] + 69.189;
   1:  PR[GP1:91,2] = PR[GP1:90,2] + 93.756;
   1:  PR[GP1:91,3] = PR[GP1:90,3] + 12.900;
   1:L PR[91] 10mm/sec FINE;
   1:  PR[GP1:91,1] = PR[GP1:90,1] + 70.688;
   1:  PR[GP1:91,2] = PR[GP1:90,2] + 93.112;
   1:L PR[91] 10mm/sec FINE;
   1:  PR[GP1:91,1] = PR[GP1:90,1] + 72.970;
   1:  PR[GP1:91,2] = PR[GP1:90,2] + 92.513;
   1:L PR[91] 10mm/sec FINE;
   1:  PR[GP1:91,1] = PR[GP1:90,1] + 74.037;
   1:  PR[GP1:91,2] = PR[GP1:90,2] + 92.301;
   1:L PR[91] 10mm/sec FINE;
   1:  PR[GP1:91,1] = PR[GP1:90,1] + 76.935;
   1:  PR[GP1:91,2] = PR[GP1:90,2] + 92.134;
   1:L PR[91] 10mm/sec FINE;
   1:  PR[GP1:91,1] = PR[GP1:90,1] + 77.402;
   1:  PR[GP1:91,2] = PR[GP1:90,2] + 92.140;
   1:L PR[91] 10mm/sec FINE;
   1:  PR[GP1:91,1] = PR[GP1:90,1] + 80.798;
   1:  PR[GP1:91,2] = PR[GP1:90,2] + 92.614;
   1:L PR[91] 10mm/sec FINE;
   1:  PR[GP1:91,1] = PR[GP1:90,1] + 83.633;
   1:  PR[GP1:91,2] = PR[GP1:90,2] + 93.558;
   1:L PR[91] 10mm/sec FINE;
   1:  PR[GP1:91,1] = PR[GP1:90,1] + 84.332;
   1:  PR[GP1:91,2] = PR[GP1:90,2] + 93.822;
   1:L PR[91] 10mm/sec FINE;
   1:  PR[GP1:91,1] = PR[GP1:90,1] + 86.385;
   1:  PR[GP1:91,2] = PR[GP1:90,2] + 95.004;
   1:L PR[91] 10mm/sec FINE;
   1:  PR[GP1:91,1] = PR[GP1:90,1] + 87.529;
   1:  PR[GP1:91,2] = PR[GP1:90,2] + 95.731;
   1:L PR[91] 10mm/sec FINE;
   1:  PR[GP1:91,1] = PR[GP1:90,1] + 88.854;
   1:  PR[GP1:91,2] = PR[GP1:90,2] + 96.912;
   1:L PR[91] 10mm/sec FINE;
   1:  PR[GP1:91,1] = PR[GP1:90,1] + 90.220;
   1:  PR[GP1:91,2] = PR[GP1:90,2] + 98.253;
   1:L PR[91] 10mm/sec FINE;
   1:  PR[GP1:91,1] = PR[GP1:90,1] + 90.975;
   1:  PR[GP1:91,2] = PR[GP1:90,2] + 99.282;
   1:L PR[91] 10mm/sec FINE;
   1:  PR[GP1:91,1] = PR[GP1:90,1] + 92.253;
   1:  PR[GP1:91,2] = PR[GP1:90,2] + 101.220;
   1:L PR[91] 10mm/sec FINE;
   1:  PR[GP1:91,1] = PR[GP1:90,1] + 92.638;
   1:  PR[GP1:91,2] = PR[GP1:90,2] + 102.061;
   1:L PR[91] 10mm/sec FINE;
   1:  PR[GP1:91,1] = PR[GP1:90,1] + 93.089;
   1:  PR[GP1:91,2] = PR[GP1:90,2] + 102.769;
   1:L PR[91] 10mm/sec FINE;
   1:  PR[GP1:91,1] = PR[GP1:90,1] + 93.260;
   1:  PR[GP1:91,2] = PR[GP1:90,2] + 102.947;
   1:L PR[91] 10mm/sec FINE;
   1:  PR[GP1:91,1] = PR[GP1:90,1] + 93.936;
   1:  PR[GP1:91,2] = PR[GP1:90,2] + 103.400;
   1:L PR[91] 10mm/sec FINE;
   1:  PR[GP1:91,1] = PR[GP1:90,1] + 94.085;
   1:  PR[GP1:91,2] = PR[GP1:90,2] + 103.444;
   1:L PR[91] 10mm/sec FINE;
   1:  PR[GP1:91,1] = PR[GP1:90,1] + 94.884;
   1:  PR[GP1:91,2] = PR[GP1:90,2] + 103.496;
   1:L PR[91] 10mm/sec FINE;
   1:  PR[GP1:91,1] = PR[GP1:90,1] + 95.020;
   1:  PR[GP1:91,2] = PR[GP1:90,2] + 103.454;
   1:L PR[91] 10mm/sec FINE;
   1:  PR[GP1:91,1] = PR[GP1:90,1] + 95.743;
   1:  PR[GP1:91,2] = PR[GP1:90,2] + 103.069;
   1:L PR[91] 10mm/sec FINE;
   1:  PR[GP1:91,1] = PR[GP1:90,1] + 95.884;
   1:  PR[GP1:91,2] = PR[GP1:90,2] + 102.913;
   1:L PR[91] 10mm/sec FINE;
   1:  PR[GP1:91,1] = PR[GP1:90,1] + 96.135;
   1:  PR[GP1:91,2] = PR[GP1:90,2] + 102.477;
   1:L PR[91] 10mm/sec FINE;
   1:  PR[GP1:91,1] = PR[GP1:90,1] + 96.326;
   1:  PR[GP1:91,2] = PR[GP1:90,2] + 102.193;
   1:L PR[91] 10mm/sec FINE;
   1:  PR[GP1:91,1] = PR[GP1:90,1] + 96.695;
   1:  PR[GP1:91,2] = PR[GP1:90,2] + 101.477;
   1:L PR[91] 10mm/sec FINE;
   1:  PR[GP1:91,1] = PR[GP1:90,1] + 97.290;
   1:  PR[GP1:91,2] = PR[GP1:90,2] + 100.404;
   1:L PR[91] 10mm/sec FINE;
   1:  PR[GP1:91,1] = PR[GP1:90,1] + 98.946;
   1:  PR[GP1:91,2] = PR[GP1:90,2] + 98.196;
   1:L PR[91] 10mm/sec FINE;
   1:  PR[GP1:91,1] = PR[GP1:90,1] + 100.870;
   1:  PR[GP1:91,2] = PR[GP1:90,2] + 96.342;
   1:L PR[91] 10mm/sec FINE;
   1:  PR[GP1:91,1] = PR[GP1:90,1] + 101.226;
   1:  PR[GP1:91,2] = PR[GP1:90,2] + 96.078;
   1:L PR[91] 10mm/sec FINE;
   1:  PR[GP1:91,1] = PR[GP1:90,1] + 103.077;
   1:  PR[GP1:91,2] = PR[GP1:90,2] + 94.786;
   1:L PR[91] 10mm/sec FINE;
   1:  PR[GP1:91,1] = PR[GP1:90,1] + 104.268;
   1:  PR[GP1:91,2] = PR[GP1:90,2] + 94.168;
   1:L PR[91] 10mm/sec FINE;
   1:  PR[GP1:91,1] = PR[GP1:90,1] + 105.522;
   1:  PR[GP1:91,2] = PR[GP1:90,2] + 93.557;
   1:L PR[91] 10mm/sec FINE;
   1:  PR[GP1:91,1] = PR[GP1:90,1] + 108.161;
   1:  PR[GP1:91,2] = PR[GP1:90,2] + 92.676;
   1:L PR[91] 10mm/sec FINE;
   1:  PR[GP1:91,1] = PR[GP1:90,1] + 111.030;
   1:  PR[GP1:91,2] = PR[GP1:90,2] + 92.137;
   1:L PR[91] 10mm/sec FINE;
   1:  PR[GP1:91,1] = PR[GP1:90,1] + 113.985;
   1:  PR[GP1:91,2] = PR[GP1:90,2] + 92.017;
   1:L PR[91] 10mm/sec FINE;
   1:  PR[GP1:91,1] = PR[GP1:90,1] + 116.905;
   1:  PR[GP1:91,2] = PR[GP1:90,2] + 92.323;
   1:L PR[91] 10mm/sec FINE;
   1:  PR[GP1:91,1] = PR[GP1:90,1] + 119.666;
   1:  PR[GP1:91,2] = PR[GP1:90,2] + 93.026;
   1:L PR[91] 10mm/sec FINE;
   1:  PR[GP1:91,1] = PR[GP1:90,1] + 122.279;
   1:  PR[GP1:91,2] = PR[GP1:90,2] + 94.127;
   1:L PR[91] 10mm/sec FINE;
   1:  PR[GP1:91,1] = PR[GP1:90,1] + 124.683;
   1:  PR[GP1:91,2] = PR[GP1:90,2] + 95.596;
   1:L PR[91] 10mm/sec FINE;
   1:  PR[GP1:91,1] = PR[GP1:90,1] + 126.822;
   1:  PR[GP1:91,2] = PR[GP1:90,2] + 97.398;
   1:L PR[91] 10mm/sec FINE;
   1:  PR[GP1:91,1] = PR[GP1:90,1] + 128.595;
   1:  PR[GP1:91,2] = PR[GP1:90,2] + 99.478;
   1:L PR[91] 10mm/sec FINE;
   1:  PR[GP1:91,1] = PR[GP1:90,1] + 130.018;
   1:  PR[GP1:91,2] = PR[GP1:90,2] + 101.801;
   1:L PR[91] 10mm/sec FINE;
   1:  PR[GP1:91,1] = PR[GP1:90,1] + 131.058;
   1:  PR[GP1:91,2] = PR[GP1:90,2] + 104.311;
   1:L PR[91] 10mm/sec FINE;
   1:  PR[GP1:91,1] = PR[GP1:90,1] + 131.692;
   1:  PR[GP1:91,2] = PR[GP1:90,2] + 106.947;
   1:L PR[91] 10mm/sec FINE;
   1:  PR[GP1:91,1] = PR[GP1:90,1] + 131.760;
   1:  PR[GP1:91,2] = PR[GP1:90,2] + 107.801;
   1:L PR[91] 10mm/sec FINE;
   1:  PR[GP1:91,1] = PR[GP1:90,1] + 131.964;
   1:  PR[GP1:91,2] = PR[GP1:90,2] + 109.652;
   1:L PR[91] 10mm/sec FINE;
   1:  PR[GP1:91,1] = PR[GP1:90,1] + 131.574;
   1:  PR[GP1:91,2] = PR[GP1:90,2] + 113.051;
   1:L PR[91] 10mm/sec FINE;
   1:  PR[GP1:91,1] = PR[GP1:90,1] + 130.553;
   1:  PR[GP1:91,2] = PR[GP1:90,2] + 116.324;
   1:L PR[91] 10mm/sec FINE;
   1:  PR[GP1:91,1] = PR[GP1:90,1] + 128.902;
   1:  PR[GP1:91,2] = PR[GP1:90,2] + 119.333;
   1:L PR[91] 10mm/sec FINE;
   1:  PR[GP1:91,1] = PR[GP1:90,1] + 126.682;
   1:  PR[GP1:91,2] = PR[GP1:90,2] + 121.961;
   1:L PR[91] 10mm/sec FINE;
   1:  PR[GP1:91,1] = PR[GP1:90,1] + 125.604;
   1:  PR[GP1:91,2] = PR[GP1:90,2] + 122.818;
   1:L PR[91] 10mm/sec FINE;
   1:  PR[GP1:91,1] = PR[GP1:90,1] + 123.946;
   1:  PR[GP1:91,2] = PR[GP1:90,2] + 124.101;
   1:L PR[91] 10mm/sec FINE;
   1:  PR[GP1:91,1] = PR[GP1:90,1] + 120.793;
   1:  PR[GP1:91,2] = PR[GP1:90,2] + 125.673;
   1:L PR[91] 10mm/sec FINE;
   1:  PR[GP1:91,1] = PR[GP1:90,1] + 117.380;
   1:  PR[GP1:91,2] = PR[GP1:90,2] + 126.617;
   1:L PR[91] 10mm/sec FINE;
   1:  PR[GP1:91,1] = PR[GP1:90,1] + 113.819;
   1:  PR[GP1:91,2] = PR[GP1:90,2] + 126.893;
   1:L PR[91] 10mm/sec FINE;
   1:  PR[GP1:91,1] = PR[GP1:90,1] + 110.194;
   1:  PR[GP1:91,2] = PR[GP1:90,2] + 126.482;
   1:L PR[91] 10mm/sec FINE;
   1:  PR[GP1:91,1] = PR[GP1:90,1] + 106.695;
   1:  PR[GP1:91,2] = PR[GP1:90,2] + 125.409;
   1:L PR[91] 10mm/sec FINE;
   1:  PR[GP1:91,1] = PR[GP1:90,1] + 103.407;
   1:  PR[GP1:91,2] = PR[GP1:90,2] + 123.702;
   1:L PR[91] 10mm/sec FINE;
   1:  PR[GP1:91,1] = PR[GP1:90,1] + 100.515;
   1:  PR[GP1:91,2] = PR[GP1:90,2] + 121.439;
   1:L PR[91] 10mm/sec FINE;
   1:  PR[GP1:91,1] = PR[GP1:90,1] + 98.124;
   1:  PR[GP1:91,2] = PR[GP1:90,2] + 118.706;
   1:L PR[91] 10mm/sec FINE;
   1:  PR[GP1:91,1] = PR[GP1:90,1] + 96.481;
   1:  PR[GP1:91,2] = PR[GP1:90,2] + 115.878;
   1:L PR[91] 10mm/sec FINE;
   1:  PR[GP1:91,1] = PR[GP1:90,1] + 95.774;
   1:  PR[GP1:91,2] = PR[GP1:90,2] + 115.020;
   1:L PR[91] 10mm/sec FINE;
   1:  PR[GP1:91,1] = PR[GP1:90,1] + 94.738;
   1:  PR[GP1:91,2] = PR[GP1:90,2] + 114.610;
   1:L PR[91] 10mm/sec FINE;
   1:  PR[GP1:91,1] = PR[GP1:90,1] + 94.448;
   1:  PR[GP1:91,2] = PR[GP1:90,2] + 114.721;
   1:L PR[91] 10mm/sec FINE;
   1:  PR[GP1:91,1] = PR[GP1:90,1] + 93.661;
   1:  PR[GP1:91,2] = PR[GP1:90,2] + 114.894;
   1:L PR[91] 10mm/sec FINE;
   1:  PR[GP1:91,1] = PR[GP1:90,1] + 93.456;
   1:  PR[GP1:91,2] = PR[GP1:90,2] + 115.133;
   1:L PR[91] 10mm/sec FINE;
   1:  PR[GP1:91,1] = PR[GP1:90,1] + 92.826;
   1:  PR[GP1:91,2] = PR[GP1:90,2] + 115.748;
   1:L PR[91] 10mm/sec FINE;
   1:  PR[GP1:91,1] = PR[GP1:90,1] + 92.660;
   1:  PR[GP1:91,2] = PR[GP1:90,2] + 116.107;
   1:L PR[91] 10mm/sec FINE;
   1:  PR[GP1:91,1] = PR[GP1:90,1] + 91.665;
   1:  PR[GP1:91,2] = PR[GP1:90,2] + 118.078;
   1:L PR[91] 10mm/sec FINE;
   1:  PR[GP1:91,1] = PR[GP1:90,1] + 91.240;
   1:  PR[GP1:91,2] = PR[GP1:90,2] + 118.656;
   1:L PR[91] 10mm/sec FINE;
   1:  PR[GP1:91,1] = PR[GP1:90,1] + 89.431;
   1:  PR[GP1:91,2] = PR[GP1:90,2] + 120.994;
   1:L PR[91] 10mm/sec FINE;
   1:  PR[GP1:91,1] = PR[GP1:90,1] + 86.961;
   1:  PR[GP1:91,2] = PR[GP1:90,2] + 123.207;
   1:L PR[91] 10mm/sec FINE;
   1:  PR[GP1:91,1] = PR[GP1:90,1] + 86.594;
   1:  PR[GP1:91,2] = PR[GP1:90,2] + 123.482;
   1:L PR[91] 10mm/sec FINE;
   1:  PR[GP1:91,1] = PR[GP1:90,1] + 84.191;
   1:  PR[GP1:91,2] = PR[GP1:90,2] + 124.909;
   1:L PR[91] 10mm/sec FINE;
   1:  PR[GP1:91,1] = PR[GP1:90,1] + 83.232;
   1:  PR[GP1:91,2] = PR[GP1:90,2] + 125.354;
   1:L PR[91] 10mm/sec FINE;
   1:  PR[GP1:91,1] = PR[GP1:90,1] + 81.074;
   1:  PR[GP1:91,2] = PR[GP1:90,2] + 126.113;
   1:L PR[91] 10mm/sec FINE;
   1:  PR[GP1:91,1] = PR[GP1:90,1] + 79.528;
   1:  PR[GP1:91,2] = PR[GP1:90,2] + 126.468;
   1:L PR[91] 10mm/sec FINE;
   1:  PR[GP1:91,1] = PR[GP1:90,1] + 77.709;
   1:  PR[GP1:91,2] = PR[GP1:90,2] + 126.725;
   1:L PR[91] 10mm/sec FINE;
   1:  PR[GP1:91,1] = PR[GP1:90,1] + 75.675;
   1:  PR[GP1:91,2] = PR[GP1:90,2] + 126.761;
   1:L PR[91] 10mm/sec FINE;
   1:  PR[GP1:91,1] = PR[GP1:90,1] + 74.224;
   1:  PR[GP1:91,2] = PR[GP1:90,2] + 126.675;
   1:L PR[91] 10mm/sec FINE;
   1:  PR[GP1:91,1] = PR[GP1:90,1] + 71.868;
   1:  PR[GP1:91,2] = PR[GP1:90,2] + 126.219;
   1:L PR[91] 10mm/sec FINE;
   1:  PR[GP1:91,1] = PR[GP1:90,1] + 70.769;
   1:  PR[GP1:91,2] = PR[GP1:90,2] + 125.929;
   1:L PR[91] 10mm/sec FINE;
   1:  PR[GP1:91,1] = PR[GP1:90,1] + 68.297;
   1:  PR[GP1:91,2] = PR[GP1:90,2] + 124.881;
   1:L PR[91] 10mm/sec FINE;
   1:  PR[GP1:91,1] = PR[GP1:90,1] + 67.502;
   1:  PR[GP1:91,2] = PR[GP1:90,2] + 124.488;
   1:L PR[91] 10mm/sec FINE;
   1:  PR[GP1:91,1] = PR[GP1:90,1] + 65.132;
   1:  PR[GP1:91,2] = PR[GP1:90,2] + 122.823;
   1:L PR[91] 10mm/sec FINE;
   1:  PR[GP1:91,1] = PR[GP1:90,1] + 64.579;
   1:  PR[GP1:91,2] = PR[GP1:90,2] + 122.394;
   1:L PR[91] 10mm/sec FINE;
   1:  PR[GP1:91,1] = PR[GP1:90,1] + 62.519;
   1:  PR[GP1:91,2] = PR[GP1:90,2] + 120.163;
   1:L PR[91] 10mm/sec FINE;
   1:  PR[GP1:91,1] = PR[GP1:90,1] + 62.145;
   1:  PR[GP1:91,2] = PR[GP1:90,2] + 119.724;
   1:L PR[91] 10mm/sec FINE;
   1:  PR[GP1:91,1] = PR[GP1:90,1] + 60.566;
   1:  PR[GP1:91,2] = PR[GP1:90,2] + 117.040;
   1:L PR[91] 10mm/sec FINE;
   1:  PR[GP1:91,1] = PR[GP1:90,1] + 60.320;
   1:  PR[GP1:91,2] = PR[GP1:90,2] + 116.595;
   1:L PR[91] 10mm/sec FINE;
   1:  PR[GP1:91,1] = PR[GP1:90,1] + 59.190;
   1:  PR[GP1:91,2] = PR[GP1:90,2] + 113.145;
   1:L PR[91] 10mm/sec FINE;
   1:  PR[GP1:91,1] = PR[GP1:90,1] + 58.874;
   1:  PR[GP1:91,2] = PR[GP1:90,2] + 110.057;
   1:L PR[91] 10mm/sec FINE;
   1:  PR[GP1:91,1] = PR[GP1:90,1] + 58.790;
   1:  PR[GP1:91,2] = PR[GP1:90,2] + 109.536;
   1:L PR[91] 10mm/sec FINE;
   1:  PR[GP1:91,1] = PR[GP1:90,1] + 59.042;
   1:  PR[GP1:91,2] = PR[GP1:90,2] + 107.272;
   1:L PR[91] 10mm/sec FINE;
   1:  PR[GP1:91,1] = PR[GP1:90,1] + 59.163;
   1:  PR[GP1:91,2] = PR[GP1:90,2] + 106.535;
   1:L PR[91] 10mm/sec FINE;
   1:  PR[GP1:91,1] = PR[GP1:90,1] + 59.233;
   1:  PR[GP1:91,2] = PR[GP1:90,2] + 105.913;
   1:L PR[91] 10mm/sec FINE;
   1:  PR[GP1:91,1] = PR[GP1:90,1] + 60.376;
   1:  PR[GP1:91,2] = PR[GP1:90,2] + 102.470;
   1:L PR[91] 10mm/sec FINE;
   1:  PR[GP1:91,1] = PR[GP1:90,1] + 60.810;
   1:  PR[GP1:91,2] = PR[GP1:90,2] + 101.699;
   1:L PR[91] 10mm/sec FINE;
   1:  PR[GP1:91,1] = PR[GP1:90,1] + 62.209;
   1:  PR[GP1:91,2] = PR[GP1:90,2] + 99.349;
   1:L PR[91] 10mm/sec FINE;
   1:  PR[GP1:91,1] = PR[GP1:90,1] + 62.959;
   1:  PR[GP1:91,2] = PR[GP1:90,2] + 98.486;
   1:L PR[91] 10mm/sec FINE;
   1:  PR[GP1:91,1] = PR[GP1:90,1] + 64.627;
   1:  PR[GP1:91,2] = PR[GP1:90,2] + 96.685;
   1:L PR[91] 10mm/sec FINE;
   1:  PR[GP1:91,1] = PR[GP1:90,1] + 65.795;
   1:  PR[GP1:91,2] = PR[GP1:90,2] + 95.787;
   1:L PR[91] 10mm/sec FINE;
   1:  PR[GP1:91,1] = PR[GP1:90,1] + 67.501;
   1:  PR[GP1:91,2] = PR[GP1:90,2] + 94.584;
   1:L PR[91] 10mm/sec FINE;
   1:  PR[GP1:91,1] = PR[GP1:90,1] + 69.854;
   1:  PR[GP1:91,2] = PR[GP1:90,2] + 93.471;
   1:  PR[GP1:91,3] = PR[GP1:90,3] + 13.900;
   1:L PR[91] 10mm/sec FINE;
   1:  PR[GP1:91,1] = PR[GP1:90,1] + 70.677;
   1:  PR[GP1:91,2] = PR[GP1:90,2] + 93.118;
   1:L PR[91] 10mm/sec FINE;
   1:  PR[GP1:91,1] = PR[GP1:90,1] + 73.680;
   1:  PR[GP1:91,2] = PR[GP1:90,2] + 92.329;
   1:L PR[91] 10mm/sec FINE;
   1:  PR[GP1:91,1] = PR[GP1:90,1] + 73.966;
   1:  PR[GP1:91,2] = PR[GP1:90,2] + 92.273;
   1:L PR[91] 10mm/sec FINE;
   1:  PR[GP1:91,1] = PR[GP1:90,1] + 77.526;
   1:  PR[GP1:91,2] = PR[GP1:90,2] + 92.052;
   1:L PR[91] 10mm/sec FINE;
   1:  PR[GP1:91,1] = PR[GP1:90,1] + 80.336;
   1:  PR[GP1:91,2] = PR[GP1:90,2] + 92.402;
   1:L PR[91] 10mm/sec FINE;
   1:  PR[GP1:91,1] = PR[GP1:90,1] + 81.256;
   1:  PR[GP1:91,2] = PR[GP1:90,2] + 92.551;
   1:L PR[91] 10mm/sec FINE;
   1:  PR[GP1:91,1] = PR[GP1:90,1] + 83.304;
   1:  PR[GP1:91,2] = PR[GP1:90,2] + 93.233;
   1:L PR[91] 10mm/sec FINE;
   1:  PR[GP1:91,1] = PR[GP1:90,1] + 84.812;
   1:  PR[GP1:91,2] = PR[GP1:90,2] + 93.804;
   1:L PR[91] 10mm/sec FINE;
   1:  PR[GP1:91,1] = PR[GP1:90,1] + 86.074;
   1:  PR[GP1:91,2] = PR[GP1:90,2] + 94.530;
   1:L PR[91] 10mm/sec FINE;
   1:  PR[GP1:91,1] = PR[GP1:90,1] + 88.018;
   1:  PR[GP1:91,2] = PR[GP1:90,2] + 95.766;
   1:L PR[91] 10mm/sec FINE;
   1:  PR[GP1:91,1] = PR[GP1:90,1] + 88.597;
   1:  PR[GP1:91,2] = PR[GP1:90,2] + 96.282;
   1:L PR[91] 10mm/sec FINE;
   1:  PR[GP1:91,1] = PR[GP1:90,1] + 90.696;
   1:  PR[GP1:91,2] = PR[GP1:90,2] + 98.343;
   1:L PR[91] 10mm/sec FINE;
   1:  PR[GP1:91,1] = PR[GP1:90,1] + 92.951;
   1:  PR[GP1:91,2] = PR[GP1:90,2] + 101.714;
   1:L PR[91] 10mm/sec FINE;
   1:  PR[GP1:91,1] = PR[GP1:90,1] + 93.322;
   1:  PR[GP1:91,2] = PR[GP1:90,2] + 102.098;
   1:L PR[91] 10mm/sec FINE;
   1:  PR[GP1:91,1] = PR[GP1:90,1] + 93.789;
   1:  PR[GP1:91,2] = PR[GP1:90,2] + 102.411;
   1:L PR[91] 10mm/sec FINE;
   1:  PR[GP1:91,1] = PR[GP1:90,1] + 94.180;
   1:  PR[GP1:91,2] = PR[GP1:90,2] + 102.528;
   1:L PR[91] 10mm/sec FINE;
   1:  PR[GP1:91,1] = PR[GP1:90,1] + 94.745;
   1:  PR[GP1:91,2] = PR[GP1:90,2] + 102.565;
   1:L PR[91] 10mm/sec FINE;
   1:  PR[GP1:91,1] = PR[GP1:90,1] + 95.125;
   1:  PR[GP1:91,2] = PR[GP1:90,2] + 102.445;
   1:L PR[91] 10mm/sec FINE;
   1:  PR[GP1:91,1] = PR[GP1:90,1] + 95.625;
   1:  PR[GP1:91,2] = PR[GP1:90,2] + 102.179;
   1:L PR[91] 10mm/sec FINE;
   1:  PR[GP1:91,1] = PR[GP1:90,1] + 95.976;
   1:  PR[GP1:91,2] = PR[GP1:90,2] + 101.793;
   1:L PR[91] 10mm/sec FINE;
   1:  PR[GP1:91,1] = PR[GP1:90,1] + 96.053;
   1:  PR[GP1:91,2] = PR[GP1:90,2] + 101.619;
   1:L PR[91] 10mm/sec FINE;
   1:  PR[GP1:91,1] = PR[GP1:90,1] + 96.654;
   1:  PR[GP1:91,2] = PR[GP1:90,2] + 100.545;
   1:L PR[91] 10mm/sec FINE;
   1:  PR[GP1:91,1] = PR[GP1:90,1] + 96.847;
   1:  PR[GP1:91,2] = PR[GP1:90,2] + 100.232;
   1:L PR[91] 10mm/sec FINE;
   1:  PR[GP1:91,1] = PR[GP1:90,1] + 98.125;
   1:  PR[GP1:91,2] = PR[GP1:90,2] + 98.507;
   1:L PR[91] 10mm/sec FINE;
   1:  PR[GP1:91,1] = PR[GP1:90,1] + 98.629;
   1:  PR[GP1:91,2] = PR[GP1:90,2] + 97.902;
   1:L PR[91] 10mm/sec FINE;
   1:  PR[GP1:91,1] = PR[GP1:90,1] + 100.252;
   1:  PR[GP1:91,2] = PR[GP1:90,2] + 96.354;
   1:L PR[91] 10mm/sec FINE;
   1:  PR[GP1:91,1] = PR[GP1:90,1] + 100.562;
   1:  PR[GP1:91,2] = PR[GP1:90,2] + 96.085;
   1:L PR[91] 10mm/sec FINE;
   1:  PR[GP1:91,1] = PR[GP1:90,1] + 102.775;
   1:  PR[GP1:91,2] = PR[GP1:90,2] + 94.567;
   1:L PR[91] 10mm/sec FINE;
   1:  PR[GP1:91,1] = PR[GP1:90,1] + 105.230;
